					IF AR3SiSortedMasterTimeBlockFreeArmBuffer[iArmFL, iFreeSlotFL, 2] > 0 THEN
					AR3SiSortedMasterTimeBlockFreeArm_Out[iArmFL, ARiFreeSlotDataQtyArm_Out[iArmFL], 1] := AR3SiSortedMasterTimeBlockFreeArmBuffer[iArmFL, iFreeSlotFL, 1];
					AR3SiSortedMasterTimeBlockFreeArm_Out[iArmFL, ARiFreeSlotDataQtyArm_Out[iArmFL], 2] := AR3SiSortedMasterTimeBlockFreeArmBuffer[iArmFL, iFreeSlotFL, 2];
					AR3SiSortedMasterTimeBlockFreeArm_Out[iArmFL, ARiFreeSlotDataQtyArm_Out[iArmFL], 3] := AR3SiSortedMasterTimeBlockFreeArmBuffer[iArmFL, iFreeSlotFL, 3];
					ARiFreeSlotDataQtyArm_Out[iArmFL] := ARiFreeSlotDataQtyArm_Out[iArmFL] +1;
					ELSE
					AR3SiSortedMasterTimeBlockFreeArm_Out[iArmFL, iFreeSlotFL, 1] := 0;
					AR3SiSortedMasterTimeBlockFreeArm_Out[iArmFL, iFreeSlotFL, 2] := 0;
					AR3SiSortedMasterTimeBlockFreeArm_Out[iArmFL, iFreeSlotFL, 3] := 0;
					END_IF

				END_IF
			END_FOR
		END_IF
	END_FOR


(*fbV2_MTBConsolidateSorted - Clear Free Slot*)

	iStnFL := 1;
	FOR iStnFL := 1 TO iStnQty DO
		IF iStnFL >= 1 AND iStnFL <= iStnQty THEN
		iFreeSlotFL := 1;
		ARiFreeSlotDataQtyStn_Out[iStnFL] := 1;
			FOR iFreeSlotFL := 1 TO ARiFreeSlotDataQtyStn_in[iStnFL] DO
				IF iFreeSlotFL >= 1 AND iFreeSlotFL <= ARiFreeSlotDataQtyStn_in[iStnFL] THEN

					IF AR3SiSortedMasterTimeBlockFreeStnBuffer[iStnFL, iFreeSlotFL, 2] > 0 THEN
					AR3SiSortedMasterTimeBlockFreeStn_Out[iStnFL, ARiFreeSlotDataQtyStn_Out[iStnFL], 1] := AR3SiSortedMasterTimeBlockFreeStnBuffer[iStnFL, iFreeSlotFL, 1];
					AR3SiSortedMasterTimeBlockFreeStn_Out[iStnFL, ARiFreeSlotDataQtyStn_Out[iStnFL], 2] := AR3SiSortedMasterTimeBlockFreeStnBuffer[iStnFL, iFreeSlotFL, 2];
					AR3SiSortedMasterTimeBlockFreeStn_Out[iStnFL, ARiFreeSlotDataQtyStn_Out[iStnFL], 3] := AR3SiSortedMasterTimeBlockFreeStnBuffer[iStnFL, iFreeSlotFL, 3];
					ARiFreeSlotDataQtyStn_Out[iStnFL] := ARiFreeSlotDataQtyStn_Out[iStnFL] +1;
					ELSE
					AR3SiSortedMasterTimeBlockFreeStn_Out[iStnFL, iFreeSlotFL, 1] := 0;
					AR3SiSortedMasterTimeBlockFreeStn_Out[iStnFL, iFreeSlotFL, 2] := 0;
					AR3SiSortedMasterTimeBlockFreeStn_Out[iStnFL, iFreeSlotFL, 3] := 0;
					END_IF

				END_IF
			END_FOR
		END_IF
	END_FOR


(*fbV2_MTBConsolidateSorted - Clear Free Slot*)

	iUldFL := 1;
	FOR iUldFL := 1 TO iUldStnQty DO
		IF iUldFL >= 1 AND iUldFL <= iUldStnQty THEN
		iFreeSlotFL := 1;
		ARiFreeSlotDataQtyUld_Out[iUldFL] := 1;
			FOR iFreeSlotFL := 1 TO ARiFreeSlotDataQtyUld_in[iUldFL] DO
				IF iFreeSlotFL >= 1 AND iFreeSlotFL <= ARiFreeSlotDataQtyUld_in[iUldFL] THEN

					IF AR3SiSortedMasterTimeBlockFreeUldBuffer[iUldFL, iFreeSlotFL, 2] > 0 THEN
					AR3SiSortedMasterTimeBlockFreeUld_Out[iUldFL, ARiFreeSlotDataQtyUld_Out[iUldFL], 1] := AR3SiSortedMasterTimeBlockFreeUldBuffer[iUldFL, iFreeSlotFL, 1];
					AR3SiSortedMasterTimeBlockFreeUld_Out[iUldFL, ARiFreeSlotDataQtyUld_Out[iUldFL], 2] := AR3SiSortedMasterTimeBlockFreeUldBuffer[iUldFL, iFreeSlotFL, 2];
					AR3SiSortedMasterTimeBlockFreeUld_Out[iUldFL, ARiFreeSlotDataQtyUld_Out[iUldFL], 3] := AR3SiSortedMasterTimeBlockFreeUldBuffer[iUldFL, iFreeSlotFL, 3];
					ARiFreeSlotDataQtyUld_Out[iUldFL] := ARiFreeSlotDataQtyUld_Out[iUldFL] +1;
					ELSE
					AR3SiSortedMasterTimeBlockFreeUld_Out[iUldFL, iFreeSlotFL, 1] := 0;
					AR3SiSortedMasterTimeBlockFreeUld_Out[iUldFL, iFreeSlotFL, 2] := 0;
					AR3SiSortedMasterTimeBlockFreeUld_Out[iUldFL, iFreeSlotFL, 3] := 0;
					END_IF

				END_IF
			END_FOR
		END_IF
	END_FOR



(*
iStep := 13;
4:
*)
	iArmFL := 1;
	FOR iArmFL := 1 TO iArmQty DO
		IF iArmFL >= 1 AND iArmFL <= iArmQty THEN
			ARiFreeSlotDataQtyArm_Out[iArmFL] := ARiFreeSlotDataQtyArm_Out[iArmFL] -1;
		END_IF
	END_FOR

	iStnFL := 1;
	FOR iStnFL := 1 TO iStnQty DO
		IF iStnFL >= 1 AND iStnFL <= iStnQty THEN
			ARiFreeSlotDataQtyStn_Out[iStnFL] := ARiFreeSlotDataQtyStn_Out[iStnFL] -1;
		END_IF
	END_FOR


	iUldFL := 1;
	FOR iUldFL := 1 TO iUldStnQty DO
		IF iUldFL >= 1 AND iUldFL <= iUldStnQty THEN
			ARiFreeSlotDataQtyUld_Out[iUldFL] := ARiFreeSlotDataQtyUld_Out[iUldFL] -1;
		END_IF
	END_FOR

(*
iStep := 14;

11:;
12:;
13:;
14:;
15:;

END_CASE
*)
bDone := TRUE;
bEn := FALSE;
iPreviousShiftValue := iShiftValue;
END_IF

END_FUNCTION_BLOCK

// ---- FBs/B_JKS_NewFB_V2/FBP-MTBSubFB/fbV2_SubMTBFreeSlotGenerator.TcPOU
FUNCTION_BLOCK fbV2_SubMTBFreeSlotGenerator


(*************************************************************** Ver.B1 - fbV2_SubMTBFreeSlotGenerator - 160704 **************************************************************]

 	- Modify Search value to 20000 from 10000. Because the Add Value when the end block will be greater than 10000.																	
	- 
	- 	
	- 
[****************************************************************************************************************************************************************************************************)



VAR_INPUT
	bReset													: BOOL;
	AR3SiMTBBusyArm_In(*AR3SiMTBArm_In*) 					: ARRAY[1..iArmQty, 1..iMasterBlockQty, 1..3] OF INT;
	AR3SiMTBBusyStn_In(*AR3SiMTBStn_In*) 					: ARRAY[1..iStnQty, 1..iMasterBlockQty, 1..3] OF INT;
	AR3SiMTBBusyUld_In(*AR3SiMTBUld_In*) 					: ARRAY[1..iUldStnQty, 1..iMasterBlockQty, 1..3] OF INT;
	ARiArmID												: ARRAY [1..iArmQty] OF INT;
	ARiUldStnID												: ARRAY [1..iUldStnQty] OF INT;		(* To Define Unloading Station ID*)


END_VAR


VAR_IN_OUT
	bEn										: BOOL;

	AR3SiSortedMTBFreeArm_Out 				: ARRAY[1..iArmQty, 1..iMasterBlockQty, 1..3] OF INT;
	AR3SiSortedMTBFreeStn_Out 				: ARRAY[1..iStnQty, 1..iMasterBlockQty, 1..3] OF INT;
	AR3SiSortedMTBFreeUld_Out 				: ARRAY[1..iUldStnQty, 1..iMasterBlockQty, 1..3] OF INT;
	ARiMTBFreeSlotDataQtyArm				: ARRAY[1..iArmQty] OF INT;
	ARiMTBFreeSlotDataQtyStn				: ARRAY[1..iStnQty] OF INT;
	ARiMTBFreeSlotDataQtyUld				: ARRAY[1..iUldStnQty] OF INT;
END_VAR

VAR_OUTPUT
	bMTBEmpty : BOOL;
	bDone : BOOL;

END_VAR
VAR
	(*AR3SiMTBArm_Out*)AR3SiSortedMTBBusyArm(*_In*) 				: ARRAY[1..iArmQty, 1..iMasterBlockQty, 1..3] OF INT;
	(*AR3SiMTBStn_Out*)AR3SiSortedMTBBusyStn(*_In*) 				: ARRAY[1..iStnQty, 1..iMasterBlockQty, 1..3] OF INT;
	(*AR3SiMTBUld_Out*)AR3SiSortedMTBBusyUld(*_In*) 				: ARRAY[1..iUldStnQty, 1..iMasterBlockQty, 1..3] OF INT;

	(*ARiDataQtyArm*)ARiSortedDataQtyArm									: ARRAY[1..iArmQty] OF INT;
	(*ARiDataQtyStn*)ARiSortedDataQtyStn									: ARRAY[1..iStnQty] OF INT;
	(*ARiDataQtyUld*)ARiSortedDataQtyUld									: ARRAY[1..iUldStnQty] OF INT;

(****** From fbV2_MTBConsolidateSorted*)
	bResetRE: R_TRIG;

	bEnRE: R_TRIG;
	bEnFE: F_TRIG;
	iStep: INT;


	AR3SiBufferTimeBlockArm 						: ARRAY[1..iArmQty, 1..iMasterBlockQty, 1..3] OF INT;
	AR3SiBufferTimeBlockStn 						: ARRAY[1..iStnQty, 1..iMasterBlockQty, 1..3] OF INT;
	AR3SiBufferTimeBlockUld 						: ARRAY[1..iUldStnQty, 1..iMasterBlockQty, 1..3] OF INT;

	AR3SiBufferOrderArm	 						: ARRAY[1..iArmQty, 1..iMasterBlockQty] OF INT;
	AR3SiBufferOrderStn 							: ARRAY[1..iStnQty, 1..iMasterBlockQty] OF INT;
	AR3SiBufferOrderUld 							: ARRAY[1..iUldStnQty, 1..iMasterBlockQty] OF INT;

	AR3SiMTBArmEmpty 				: ARRAY[1..iArmQty, 1..iMasterBlockQty, 1..3] OF INT;
	AR3SiMTBStnEmpty 				: ARRAY[1..iStnQty, 1..iMasterBlockQty, 1..3] OF INT;
	AR3SiMTBUldEmpty 				: ARRAY[1..iUldStnQty, 1..iMasterBlockQty, 1..3] OF INT;

	AR3SiBufferOrderArmEmpty	 				: ARRAY[1..iArmQty, 1..iMasterBlockQty] OF INT;
	AR3SiBufferOrderStnEmpty	 					: ARRAY[1..iStnQty, 1..iMasterBlockQty] OF INT;
	AR3SiBufferOrderUldEmpty	 					: ARRAY[1..iUldStnQty, 1..iMasterBlockQty] OF INT;


	ARiCounterArmEmpty: ARRAY[1..iArmQty] OF INT;
	ARiCounterStnEmpty: ARRAY[1..iStnQty] OF INT;
	ARiCounterUldEmpty: ARRAY[1..iUldStnQty] OF INT;

	iSearchFL: INT;
	iSearchBuffer: INT;
	iSearchBufferAdd: INT;
	iSearchBufferValue: INT;
	iCounter: INT;
	iRunningNo: INT;

	iCheckFL: INT;
	iFreeSlotFL: INT;

	iArmFL: INT;
	iStnFL: INT;
	iUldFL: INT;

	ARiFoundCounterArm: ARRAY[1..iArmQty] OF INT;
	ARiFoundCounterStn: ARRAY[1..iStnQty] OF INT;
	ARiFoundCounterUld: ARRAY[1..iUldStnQty] OF INT;

	ARiScanCounterArm: ARRAY[1..iArmQty] OF INT;
	ARiScanCounterStn: ARRAY[1..iStnQty] OF INT;
	ARiScanCounterUld: ARRAY[1..iUldStnQty] OF INT;


	iGenFL: INT;
	iSkipArm: INT;
	iSkipStn: INT;
	iSkipUld: INT;
END_VAR

bResetRE(CLK:=bReset , Q=> );
bEnRE(CLK:=bEn , Q=> );

IF bResetRE.Q THEN
bDone := FALSE;
bMTBEmpty := FALSE;
END_IF

(*
IF NOT bEn THEN
bDone := FALSE;
END_IF
*)


IF NOT bReset AND bEnRE.Q THEN

	bDone := FALSE;
	bMTBEmpty := FALSE;
	iStep := 1;
	AR3SiSortedMTBBusyArm 				:= AR3SiMTBArmEmpty;
	AR3SiSortedMTBBusyStn 				:= AR3SiMTBStnEmpty;
	AR3SiSortedMTBBusyUld 				:= AR3SiMTBUldEmpty;

	AR3SiBufferOrderArm 					:= AR3SiBufferOrderArmEmpty;
	AR3SiBufferOrderStn 					:= AR3SiBufferOrderStnEmpty;
	AR3SiBufferOrderUld 					:= AR3SiBufferOrderUldEmpty;

	AR3SiBufferTimeBlockArm 				:= AR3SiMTBArmEmpty;
	AR3SiBufferTimeBlockStn 				:= AR3SiMTBStnEmpty;
	AR3SiBufferTimeBlockUld 				:= AR3SiMTBUldEmpty;

	ARiSortedDataQtyArm 					:= ARiCounterArmEmpty;
	ARiSortedDataQtyStn 					:= ARiCounterStnEmpty;
	ARiSortedDataQtyUld					:= ARiCounterUldEmpty;

	AR3SiSortedMTBFreeArm_Out 			:= AR3SiMTBArmEmpty;
	AR3SiSortedMTBFreeStn_Out 			:= AR3SiMTBStnEmpty;
	AR3SiSortedMTBFreeUld_Out 			:= AR3SiMTBUldEmpty;



END_IF

CASE iStep OF
0:;

1: (*fbV2_MTBConsolidateSorted - Clear Free Slot*)
	iArmFL := 1;
	FOR iArmFL := 1 TO iArmQty DO
		IF iArmFL >= 1 AND iArmFL <= iArmQty THEN
		iFreeSlotFL := 1;
		ARiSortedDataQtyArm[iArmFL] := 1;
			FOR iFreeSlotFL := 1 TO iMasterBlockQty DO
				IF iFreeSlotFL >= 1 AND iFreeSlotFL <= iMasterBlockQty THEN

					IF AR3SiMTBBusyArm_In[iArmFL, iFreeSlotFL, 2] > 0 THEN
					AR3SiBufferTimeBlockArm[iArmFL, ARiSortedDataQtyArm[iArmFL], 1] := AR3SiMTBBusyArm_In[iArmFL, iFreeSlotFL, 1];
					AR3SiBufferTimeBlockArm[iArmFL, ARiSortedDataQtyArm[iArmFL], 2] := AR3SiMTBBusyArm_In[iArmFL, iFreeSlotFL, 2];
					AR3SiBufferTimeBlockArm[iArmFL, ARiSortedDataQtyArm[iArmFL], 3] := AR3SiMTBBusyArm_In[iArmFL, iFreeSlotFL, 3];
					ARiSortedDataQtyArm[iArmFL] := ARiSortedDataQtyArm[iArmFL] +1;
					END_IF
				END_IF
			END_FOR
		END_IF
	END_FOR


	iStnFL := 1;
	FOR iStnFL := 1 TO iStnQty DO
		IF iStnFL >= 1 AND iStnFL <= iStnQty THEN
		iFreeSlotFL := 1;
		ARiSortedDataQtyStn[iStnFL] := 1;
			FOR iFreeSlotFL := 1 TO iMasterBlockQty DO
				IF iFreeSlotFL >= 1 AND iFreeSlotFL <= iMasterBlockQty THEN

					IF AR3SiMTBBusyStn_In[iStnFL, iFreeSlotFL, 2] > 0 THEN
					AR3SiBufferTimeBlockStn[iStnFL, ARiSortedDataQtyStn[iStnFL], 1] := AR3SiMTBBusyStn_In[iStnFL, iFreeSlotFL, 1];
					AR3SiBufferTimeBlockStn[iStnFL, ARiSortedDataQtyStn[iStnFL], 2] := AR3SiMTBBusyStn_In[iStnFL, iFreeSlotFL, 2];
					AR3SiBufferTimeBlockStn[iStnFL, ARiSortedDataQtyStn[iStnFL], 3] := AR3SiMTBBusyStn_In[iStnFL, iFreeSlotFL, 3];
					ARiSortedDataQtyStn[iStnFL] := ARiSortedDataQtyStn[iStnFL] +1;
					END_IF
				END_IF
			END_FOR
		END_IF
	END_FOR



	iUldFL := 1;
	FOR iUldFL := 1 TO iUldStnQty DO
		IF iUldFL >= 1 AND iUldFL <= iUldStnQty THEN
		iFreeSlotFL := 1;
		ARiSortedDataQtyUld[iUldFL] := 1;
			FOR iFreeSlotFL := 1 TO iMasterBlockQty DO
				IF iFreeSlotFL >= 1 AND iFreeSlotFL <= iMasterBlockQty THEN

					IF AR3SiMTBBusyUld_In[iUldFL, iFreeSlotFL, 2] > 0 THEN
					AR3SiBufferTimeBlockUld[iUldFL, ARiSortedDataQtyUld[iUldFL], 1] := AR3SiMTBBusyUld_In[iUldFL, iFreeSlotFL, 1];
					AR3SiBufferTimeBlockUld[iUldFL, ARiSortedDataQtyUld[iUldFL], 2] := AR3SiMTBBusyUld_In[iUldFL, iFreeSlotFL, 2];
					AR3SiBufferTimeBlockUld[iUldFL, ARiSortedDataQtyUld[iUldFL], 3] := AR3SiMTBBusyUld_In[iUldFL, iFreeSlotFL, 3];
					ARiSortedDataQtyUld[iUldFL] := ARiSortedDataQtyUld[iUldFL] +1;
					END_IF
				END_IF
			END_FOR
		END_IF
	END_FOR



	iArmFL := 1;
	FOR iArmFL := 1 TO iArmQty DO
		IF iArmFL >= 1 AND iArmFL <= iArmQty THEN
			ARiSortedDataQtyArm[iArmFL] := ARiSortedDataQtyArm[iArmFL] -1;
			ARiMTBFreeSlotDataQtyArm[iArmFL] := 0;
		END_IF
	END_FOR

	iStnFL := 1;
	FOR iStnFL := 1 TO iStnQty DO
		IF iStnFL >= 1 AND iStnFL <= iStnQty THEN
			ARiSortedDataQtyStn[iStnFL] := ARiSortedDataQtyStn[iStnFL] -1;
			ARiMTBFreeSlotDataQtyStn[iStnFL] := 0;
		END_IF
	END_FOR

	iUldFL := 1;
	FOR iUldFL := 1 TO iUldStnQty DO
		IF iUldFL >= 1 AND iUldFL <= iUldStnQty THEN
			ARiSortedDataQtyUld[iUldFL] := ARiSortedDataQtyUld[iUldFL] -1;
			ARiMTBFreeSlotDataQtyUld[iUldFL] := 0;
		END_IF
	END_FOR




iArmFL := 1;
iStnFL := 1;
iUldFL := 1;



iStep := 12;



12: (*fbV2_MTBConsolidateSorted - Data Sorting*)

	IF iArmFL <= iArmQty THEN
		ARiScanCounterArm[iArmFL] := 1;
		ARiFoundCounterArm[iArmFL] := 1;

		FOR ARiScanCounterArm[iArmFL] := 1 TO ARiSortedDataQtyArm[iArmFL] DO
			IF ARiScanCounterArm[iArmFL] >= 1 AND ARiScanCounterArm[iArmFL] <= ARiSortedDataQtyArm[iArmFL] THEN

				iSearchFL := 1;
				iSearchBufferValue := 20000;
				iSearchBufferAdd := 0;
					FOR iSearchFL := 1 TO ARiSortedDataQtyArm[iArmFL] DO
						IF iSearchFL >= 1 AND iSearchFL <= ARiSortedDataQtyArm[iArmFL] THEN

							IF AR3SiBufferOrderArm[iArmFL, iSearchFL] = 0 AND AR3SiBufferTimeBlockArm[iArmFL, iSearchFL, 2] > 0 THEN
								IF AR3SiBufferTimeBlockArm[iArmFL, iSearchFL, 2] <= iSearchBufferValue THEN
									iSearchBufferValue		:= AR3SiBufferTimeBlockArm[iArmFL, iSearchFL, 2];
									iSearchBufferAdd			:= iSearchFL;
								END_IF
							END_IF
						END_IF

					END_FOR

					IF iSearchFL > ARiSortedDataQtyArm[iArmFL] AND iSearchBufferAdd > 0 THEN
					AR3SiSortedMTBBusyArm[iArmFL, ARiFoundCounterArm[iArmFL], 1] := AR3SiBufferTimeBlockArm[iArmFL, iSearchBufferAdd, 1];
					AR3SiSortedMTBBusyArm[iArmFL, ARiFoundCounterArm[iArmFL], 2] := AR3SiBufferTimeBlockArm[iArmFL, iSearchBufferAdd, 2];
					AR3SiSortedMTBBusyArm[iArmFL, ARiFoundCounterArm[iArmFL], 3] := AR3SiBufferTimeBlockArm[iArmFL, iSearchBufferAdd, 3];
					AR3SiBufferOrderArm[iArmFL, iSearchBufferAdd] := ARiFoundCounterArm[iArmFL];
					ARiFoundCounterArm[iArmFL] := ARiFoundCounterArm[iArmFL] +1;
					END_IF

			END_IF
		END_FOR
	END_IF



	IF iStnFL <= iStnQty THEN
		ARiScanCounterStn[iStnFL] := 1;
		ARiFoundCounterStn[iStnFL] := 1;

		FOR ARiScanCounterStn[iStnFL] := 1 TO ARiSortedDataQtyStn[iStnFL] DO
			IF ARiScanCounterStn[iStnFL] >= 1 AND ARiScanCounterStn[iStnFL] <= ARiSortedDataQtyStn[iStnFL] THEN

				iSearchFL := 1;
				iSearchBufferValue := 20000;
				iSearchBufferAdd := 0;
					FOR iSearchFL := 1 TO ARiSortedDataQtyStn[iStnFL] DO
						IF iSearchFL >= 1 AND iSearchFL <= ARiSortedDataQtyStn[iStnFL] THEN

							IF AR3SiBufferOrderStn[iStnFL, iSearchFL] = 0 AND AR3SiBufferTimeBlockStn[iStnFL, iSearchFL, 2] > 0 THEN
								IF AR3SiBufferTimeBlockStn[iStnFL, iSearchFL, 2] <= iSearchBufferValue THEN
									iSearchBufferValue		:= AR3SiBufferTimeBlockStn[iStnFL, iSearchFL, 2];
									iSearchBufferAdd			:= iSearchFL;
								END_IF
							END_IF
						END_IF

					END_FOR

					IF iSearchFL > ARiSortedDataQtyStn[iStnFL] AND iSearchBufferAdd > 0 THEN
					AR3SiSortedMTBBusyStn[iStnFL, ARiFoundCounterStn[iStnFL], 1] := AR3SiBufferTimeBlockStn[iStnFL, iSearchBufferAdd, 1];
					AR3SiSortedMTBBusyStn[iStnFL, ARiFoundCounterStn[iStnFL], 2] := AR3SiBufferTimeBlockStn[iStnFL, iSearchBufferAdd, 2];
					AR3SiSortedMTBBusyStn[iStnFL, ARiFoundCounterStn[iStnFL], 3] := AR3SiBufferTimeBlockStn[iStnFL, iSearchBufferAdd, 3];
					AR3SiBufferOrderStn[iStnFL, iSearchBufferAdd] := ARiFoundCounterStn[iStnFL];
					ARiFoundCounterStn[iStnFL] := ARiFoundCounterStn[iStnFL] +1;
					END_IF

			END_IF
		END_FOR
	END_IF



	IF iUldFL <= iUldStnQty THEN
		ARiScanCounterUld[iUldFL] := 1;
		ARiFoundCounterUld[iUldFL] := 1;

		FOR ARiScanCounterUld[iUldFL] := 1 TO ARiSortedDataQtyUld[iUldFL] DO
			IF ARiScanCounterUld[iUldFL] >= 1 AND ARiScanCounterUld[iUldFL] <= ARiSortedDataQtyUld[iUldFL] THEN

				iSearchFL := 1;
				iSearchBufferValue := 20000;
				iSearchBufferAdd := 0;
					FOR iSearchFL := 1 TO ARiSortedDataQtyUld[iUldFL] DO
						IF iSearchFL >= 1 AND iSearchFL <= ARiSortedDataQtyUld[iUldFL] THEN

							IF AR3SiBufferOrderUld[iUldFL, iSearchFL] = 0 AND AR3SiBufferTimeBlockUld[iUldFL, iSearchFL, 2] > 0 THEN
								IF AR3SiBufferTimeBlockUld[iUldFL, iSearchFL, 2] <= iSearchBufferValue THEN
									iSearchBufferValue		:= AR3SiBufferTimeBlockUld[iUldFL, iSearchFL, 2];
									iSearchBufferAdd			:= iSearchFL;
								END_IF
							END_IF
						END_IF

					END_FOR

					IF iSearchFL > ARiSortedDataQtyUld[iUldFL] AND iSearchBufferAdd > 0 THEN
					AR3SiSortedMTBBusyUld[iUldFL, ARiFoundCounterUld[iUldFL], 1] := AR3SiBufferTimeBlockUld[iUldFL, iSearchBufferAdd, 1];
					AR3SiSortedMTBBusyUld[iUldFL, ARiFoundCounterUld[iUldFL], 2] := AR3SiBufferTimeBlockUld[iUldFL, iSearchBufferAdd, 2];
					AR3SiSortedMTBBusyUld[iUldFL, ARiFoundCounterUld[iUldFL], 3] := AR3SiBufferTimeBlockUld[iUldFL, iSearchBufferAdd, 3];
					AR3SiBufferOrderUld[iUldFL, iSearchBufferAdd] := ARiFoundCounterUld[iUldFL];
					ARiFoundCounterUld[iUldFL] := ARiFoundCounterUld[iUldFL] +1;
					END_IF

			END_IF
		END_FOR
	END_IF

iArmFL := iArmFL +1;
iStnFL := iStnFL +1;
iUldFL := iUldFL +1;

IF iArmFL > iArmQty AND iStnFL > iStnQty AND iUldFL > iUldStnQty THEN
iStep := 13;
END_IF

13:(*Generate FreeSlotBlock from Busy Block*)

	iArmFL := 1;
	iStnFL := 1;
	iUldFL := 1;

	FOR iArmFL := 1 TO iArmQty DO
		IF iArmFL >= 1 AND iArmFL <= iArmQty THEN
			iGenFL := 1;
			iSkipArm := 0;
			FOR iGenFL := 1 TO ARiSortedDataQtyArm[iArmFL] DO
				IF iGenFL >= 1 AND iGenFL <= ARiSortedDataQtyArm[iArmFL] THEN

					IF iGenFL = 1 THEN
						IF AR3SiSortedMTBBusyArm[iArmFL, iGenFL, 1] >1(*0*) THEN
							AR3SiSortedMTBFreeArm_Out[iArmFL, iGenFL, 1] := 0;
							AR3SiSortedMTBFreeArm_Out[iArmFL, iGenFL, 2] := AR3SiSortedMTBBusyArm[iArmFL, iGenFL, 1]-1;
							AR3SiSortedMTBFreeArm_Out[iArmFL, iGenFL, 3] := AR3SiSortedMTBBusyArm[iArmFL, iGenFL, 3];
							ARiMTBFreeSlotDataQtyArm[iArmFL] := ARiMTBFreeSlotDataQtyArm[iArmFL] +1;
						ELSE
							iSkipArm := 1;
						END_IF
					END_IF

					IF iGenFL >1 THEN
						IF AR3SiSortedMTBBusyArm[iArmFL, iGenFL, 1] >1(*0*) THEN
							AR3SiSortedMTBFreeArm_Out[iArmFL, iGenFL-iSkipArm, 1] := AR3SiSortedMTBBusyArm[iArmFL, iGenFL-1, 2]+1;
							AR3SiSortedMTBFreeArm_Out[iArmFL, iGenFL-iSkipArm, 2] := AR3SiSortedMTBBusyArm[iArmFL, iGenFL, 1]-1;
							AR3SiSortedMTBFreeArm_Out[iArmFL, iGenFL-iSkipArm, 3] := AR3SiSortedMTBBusyArm[iArmFL, iGenFL, 3];
							ARiMTBFreeSlotDataQtyArm[iArmFL] := ARiMTBFreeSlotDataQtyArm[iArmFL] +1;
						END_IF
					END_IF

					IF iGenFL =ARiSortedDataQtyArm[iArmFL] THEN
						IF AR3SiSortedMTBBusyArm[iArmFL, iGenFL, 2] >1(*0*) THEN
							AR3SiSortedMTBFreeArm_Out[iArmFL, iGenFL-iSkipArm+1, 1] := AR3SiSortedMTBBusyArm[iArmFL, iGenFL, 2]+1;
							AR3SiSortedMTBFreeArm_Out[iArmFL, iGenFL-iSkipArm+1, 2] := AR3SiSortedMTBBusyArm[iArmFL, iGenFL, 2]+1+10000;
							AR3SiSortedMTBFreeArm_Out[iArmFL, iGenFL-iSkipArm+1, 3] := AR3SiSortedMTBBusyArm[iArmFL, iGenFL, 3];
							ARiMTBFreeSlotDataQtyArm[iArmFL] := ARiMTBFreeSlotDataQtyArm[iArmFL] +1;
						END_IF
					END_IF
				END_IF
			END_FOR
		END_IF
	END_FOR


	FOR iStnFL := 1 TO iStnQty DO
		IF iStnFL >= 1 AND iStnFL <= iStnQty THEN
			iGenFL := 1;
			iSkipStn := 0;
			FOR iGenFL := 1 TO ARiSortedDataQtyStn[iStnFL] DO
				IF iGenFL >= 1 AND iGenFL <= ARiSortedDataQtyStn[iStnFL] THEN

					IF iGenFL = 1 THEN
						IF AR3SiSortedMTBBusyStn[iStnFL, iGenFL, 1] >1(*0*) THEN
							AR3SiSortedMTBFreeStn_Out[iStnFL, iGenFL, 1] := 0;
							AR3SiSortedMTBFreeStn_Out[iStnFL, iGenFL, 2] := AR3SiSortedMTBBusyStn[iStnFL, iGenFL, 1]-1;
							AR3SiSortedMTBFreeStn_Out[iStnFL, iGenFL, 3] := AR3SiSortedMTBBusyStn[iStnFL, iGenFL, 3];
							ARiMTBFreeSlotDataQtyStn[iStnFL] := ARiMTBFreeSlotDataQtyStn[iStnFL] +1;
						ELSE
							iSkipStn := 1;
						END_IF
					END_IF

					IF iGenFL >1 THEN
						IF AR3SiSortedMTBBusyStn[iStnFL, iGenFL, 1] >1(*0*) THEN
							AR3SiSortedMTBFreeStn_Out[iStnFL, iGenFL-iSkipStn, 1] := AR3SiSortedMTBBusyStn[iStnFL, iGenFL-1, 2]+1;
							AR3SiSortedMTBFreeStn_Out[iStnFL, iGenFL-iSkipStn, 2] := AR3SiSortedMTBBusyStn[iStnFL, iGenFL, 1]-1;
							AR3SiSortedMTBFreeStn_Out[iStnFL, iGenFL-iSkipStn, 3] := AR3SiSortedMTBBusyStn[iStnFL, iGenFL, 3];
							ARiMTBFreeSlotDataQtyStn[iStnFL] := ARiMTBFreeSlotDataQtyStn[iStnFL] +1;
						END_IF
					END_IF

					IF iGenFL =ARiSortedDataQtyStn[iStnFL] THEN
						IF AR3SiSortedMTBBusyStn[iStnFL, iGenFL, 2] >1(*0*) THEN
							AR3SiSortedMTBFreeStn_Out[iStnFL, iGenFL-iSkipStn+1, 1] := AR3SiSortedMTBBusyStn[iStnFL, iGenFL, 2]+1;
							AR3SiSortedMTBFreeStn_Out[iStnFL, iGenFL-iSkipStn+1, 2] := AR3SiSortedMTBBusyStn[iStnFL, iGenFL, 2]+1+10000;
							AR3SiSortedMTBFreeStn_Out[iStnFL, iGenFL-iSkipStn+1, 3] := AR3SiSortedMTBBusyStn[iStnFL, iGenFL, 3];
							ARiMTBFreeSlotDataQtyStn[iStnFL] := ARiMTBFreeSlotDataQtyStn[iStnFL] +1;
						END_IF
					END_IF
				END_IF
			END_FOR
		END_IF
	END_FOR



	FOR iUldFL := 1 TO iUldStnQty DO
		IF iUldFL >= 1 AND iUldFL <= iUldStnQty THEN
			iGenFL := 1;
			iSkipUld := 0;
			FOR iGenFL := 1 TO ARiSortedDataQtyUld[iUldFL] DO
				IF iGenFL >= 1 AND iGenFL <= ARiSortedDataQtyUld[iUldFL] THEN

					IF iGenFL = 1 THEN
						IF AR3SiSortedMTBBusyUld[iUldFL, iGenFL, 1] >1(*0*) THEN
							AR3SiSortedMTBFreeUld_Out[iUldFL, iGenFL, 1] := 0;
							AR3SiSortedMTBFreeUld_Out[iUldFL, iGenFL, 2] := AR3SiSortedMTBBusyUld[iUldFL, iGenFL, 1]-1;
							AR3SiSortedMTBFreeUld_Out[iUldFL, iGenFL, 3] := AR3SiSortedMTBBusyUld[iUldFL, iGenFL, 3];
							ARiMTBFreeSlotDataQtyUld[iUldFL] := ARiMTBFreeSlotDataQtyUld[iUldFL] +1;
						ELSE
							iSkipUld := 1;
						END_IF
					END_IF

					IF iGenFL >1 THEN
						IF AR3SiSortedMTBBusyUld[iUldFL, iGenFL, 1] >1(*0*) THEN
							AR3SiSortedMTBFreeUld_Out[iUldFL, iGenFL-iSkipUld, 1] := AR3SiSortedMTBBusyUld[iUldFL, iGenFL-1, 2]+1;
							AR3SiSortedMTBFreeUld_Out[iUldFL, iGenFL-iSkipUld, 2] := AR3SiSortedMTBBusyUld[iUldFL, iGenFL, 1]-1;
							AR3SiSortedMTBFreeUld_Out[iUldFL, iGenFL-iSkipUld, 3] := AR3SiSortedMTBBusyUld[iUldFL, iGenFL, 3];
							ARiMTBFreeSlotDataQtyUld[iUldFL] := ARiMTBFreeSlotDataQtyUld[iUldFL] +1;
						END_IF
					END_IF

					IF iGenFL =ARiSortedDataQtyUld[iUldFL] THEN
						IF AR3SiSortedMTBBusyUld[iUldFL, iGenFL, 2] >1(*0*) THEN
							AR3SiSortedMTBFreeUld_Out[iUldFL, iGenFL-iSkipUld+1, 1] := AR3SiSortedMTBBusyUld[iUldFL, iGenFL, 2]+1;
							AR3SiSortedMTBFreeUld_Out[iUldFL, iGenFL-iSkipUld+1, 2] := AR3SiSortedMTBBusyUld[iUldFL, iGenFL, 2]+1+10000;
							AR3SiSortedMTBFreeUld_Out[iUldFL, iGenFL-iSkipUld+1, 3] := AR3SiSortedMTBBusyUld[iUldFL, iGenFL, 3];
							ARiMTBFreeSlotDataQtyUld[iUldFL] := ARiMTBFreeSlotDataQtyUld[iUldFL] +1;
						END_IF
					END_IF
				END_IF
			END_FOR
		END_IF
	END_FOR




iStep:= 14;

14: (* Put Remark for those "0" = "Empty" Stn *) (*Generate FreeSlotBlock for Empty Stn Block*)

bMTBEmpty := TRUE;

	iArmFL := 1;
	FOR iArmFL := 1 TO iArmQty DO
		IF iArmFL >= 1 AND iArmFL <= iArmQty THEN

			IF ARiMTBFreeSlotDataQtyArm[iArmFL] > 0 THEN
				bMTBEmpty := FALSE;
			END_IF

			IF ARiMTBFreeSlotDataQtyArm[iArmFL] = 0 THEN
				AR3SiSortedMTBFreeArm_Out[iArmFL, 1, 1] := 0;
				AR3SiSortedMTBFreeArm_Out[iArmFL, 1, 2] := 10000;
				AR3SiSortedMTBFreeArm_Out[iArmFL, 1, 3] := ARiArmID[iArmFL];
				ARiMTBFreeSlotDataQtyArm[iArmFL] := 1;
			END_IF
		END_IF
	END_FOR


	iStnFL := 1;
	FOR iStnFL := 1 TO iStnQty DO
		IF iStnFL >= 1 AND iStnFL <= iStnQty THEN

			IF ARiMTBFreeSlotDataQtyStn[iStnFL] > 0 THEN
				bMTBEmpty := FALSE;
			END_IF

			IF ARiMTBFreeSlotDataQtyStn[iStnFL] = 0 THEN
				AR3SiSortedMTBFreeStn_Out[iStnFL, 1, 1] := 0;
				AR3SiSortedMTBFreeStn_Out[iStnFL, 1, 2] := 10000;
				AR3SiSortedMTBFreeStn_Out[iStnFL, 1, 3] := iStnFL;
				ARiMTBFreeSlotDataQtyStn[iStnFL] := 1;
			END_IF
		END_IF
	END_FOR


	iUldFL := 1;
	FOR iUldFL := 1 TO iUldStnQty DO
		IF iUldFL >= 1 AND iUldFL <= iUldStnQty THEN

			IF ARiMTBFreeSlotDataQtyUld[iUldFL] > 0 THEN
				bMTBEmpty := FALSE;
			END_IF

			IF ARiMTBFreeSlotDataQtyUld[iUldFL] = 0 THEN
				AR3SiSortedMTBFreeUld_Out[iUldFL, 1, 1] := 0;
				AR3SiSortedMTBFreeUld_Out[iUldFL, 1, 2] := 10000;
				AR3SiSortedMTBFreeUld_Out[iUldFL, 1, 3] := ARiUldStnID[iUldFL];
				ARiMTBFreeSlotDataQtyUld[iUldFL] := 1;
			END_IF
		END_IF
	END_FOR

iStep := 20;


20: (* Search Completed*)
bDone := TRUE;
bEn := FALSE;


END_CASE

END_FUNCTION_BLOCK

// ---- FBs/B_JKS_NewFB_V2/FBP-MTBSubFB/fbV2_SubMTBRTBCrashCheck.TcPOU
FUNCTION_BLOCK fbV2_SubMTBRTBCrashCheck
VAR_INPUT
	bEn										: BOOL;
	bReset									: BOOL;
	bBusyLinkMasterCheck					: BOOL;
	bBusyLinkSlaveCheck						: BOOL;
	iCurrentMasterFreeBlockStart 				: INT; 	(*MD1*)		(*Array "1"*)
	iCurrentMasterFreeBlockEnd 				: INT;	(*MD2*)		(*Array "2"*)
(*	iNextMasterFreeBlockStart 					: INT; 	(*MD3*)
	iNextMasterFreeBlockEnd 					: INT;	(*MD4*)
*)	iCurrentRecipeBusyBlockStart 				: INT;	(*RD1*)		(*Array "1"*)
	iCurrentRecipeBusyBlockEnd 				: INT;	(*RD2*)		(*Array "2"*)
	iCurrentRecipeBusyTime					: INT;				(*Array "5"*)
	iCurrentRecipeBusyBlockMinTime			: INT;				(*Array "6"*)
	iCurrentRecipeBusyBlockMaxTime			: INT;				(*Array "7"*)
	iCurrentRecipeBusyLinkMasterSlaveAdd		: INT;				(*Array "9"*)
	iCurrentShiftAllowedTime					: INT; 	(*Determine by Previous Station Remained Tolerance Time VS Crashed Time Whichever Lower*)

END_VAR
VAR_IN_OUT
	iMTB_NATime							: INT;
END_VAR

VAR_OUTPUT

(**)	bMTB_ShiftBlockRequestFlag	: BOOL; (*Current Master Time Block Empty or Not Suitable for Scanning Used, Out of range*)
(**)	bRTB_ShiftBlockRequestFlag	: BOOL; (*Current Recipe Time Block Empty*)
(**)	bSpacingOK 					: BOOL;
(**)	bNoCrashFound				: BOOL;
(**)	iNextShiftAllowedTime			: INT;	(*Determine Balance Time for Next Block Shifting Based on Remained Tolerance Time VS Crashed Time whichever lower*)

(**)	bSpacingNG 					: BOOL;
	bCrashFound 				: BOOL;

(**)	bMTB_ShiftTimeRequestFlag 	: BOOL;
(**)	iMTB_ShiftTime	 			: INT;

(**)	bRTB_ShiftTimeRequestFlag 	: BOOL;
(**)	iRTB_ShiftTime	 			: INT;

	bBusyLinkMasterSkipFlag		: BOOL;
	bBusyLinkSlaveSkipFlag		: BOOL;

	bError						: BOOL;


END_VAR
VAR

	bEnFE: F_TRIG;
	iCurrentRecipeBusyBlockTolerance	: INT;

	iExtTime: INT;
	bResetRE: R_TRIG;
END_VAR

bResetRE(CLK:=bReset , Q=> );

IF bResetRE.Q THEN
	bMTB_ShiftBlockRequestFlag	:= FALSE;
	bRTB_ShiftBlockRequestFlag	:= FALSE;

	bSpacingOK 					:= FALSE;
	bNoCrashFound				:= FALSE;
	iNextShiftAllowedTime 			:= 0;

	bSpacingNG 					:= FALSE;
	bCrashFound 				:= FALSE;

	bMTB_ShiftTimeRequestFlag 	:= FALSE;
	iMTB_ShiftTime	 			:= 0;

	bRTB_ShiftTimeRequestFlag 	:= FALSE;
	iRTB_ShiftTime	 			:= 0;

	bBusyLinkMasterSkipFlag		:= FALSE;
	bBusyLinkSlaveSkipFlag		:= FALSE;
	bError						:= FALSE;

END_IF


IF bEn THEN

(*Initialised*)
	bMTB_ShiftBlockRequestFlag	:= FALSE;
	bRTB_ShiftBlockRequestFlag	:= FALSE;

	bSpacingOK 					:= FALSE;
	bNoCrashFound				:= FALSE;
	iNextShiftAllowedTime 			:= 0;

	bSpacingNG 					:= FALSE;
	bCrashFound 				:= FALSE;

	bMTB_ShiftTimeRequestFlag 	:= FALSE;
	iMTB_ShiftTime	 			:= 0;

	bRTB_ShiftTimeRequestFlag 	:= FALSE;
	iRTB_ShiftTime	 			:= 0;

	bBusyLinkMasterSkipFlag		:= FALSE;
	bBusyLinkSlaveSkipFlag		:= FALSE;
	bError						:= FALSE;



(*Checking / Scanning Start*)

	(*Check BusyLink Master And Slave Operation*)
	IF bBusyLinkMasterCheck AND iCurrentRecipeBusyLinkMasterSlaveAdd > 99 THEN
		bBusyLinkSlaveSkipFlag := TRUE;
	ELSIF bBusyLinkSlaveCheck AND iCurrentRecipeBusyLinkMasterSlaveAdd <100 THEN
		bBusyLinkMasterSkipFlag := TRUE;

	(*RTB Empty / Error Block - Cannot Scan*)
	ELSIF (iCurrentRecipeBusyBlockEnd (*RD2*)  <= 0)									(*Empty Block*)
		OR (iCurrentRecipeBusyBlockStart (*RD1*) >= iCurrentRecipeBusyBlockEnd (*RD2*))	(*Error Block*)
		THEN

		bRTB_ShiftBlockRequestFlag	:= TRUE;
		bError						:= TRUE;


	(*MTB Empty / Error - Cannot Scan*)

	ELSIF (iCurrentMasterFreeBlockEnd (*MD2*)  <= 0)									(*Empty Block*)
		OR( (iCurrentMasterFreeBlockStart (*MD1*) ) - (iCurrentMasterFreeBlockEnd (*MD2*))) > 1		(*Error Block*)
		(*OR (iCurrentMasterFreeBlockEnd (*MD2*) <= iCurrentRecipeBusyBlockStart (*RD1*))		(*Not Suitable Block*)*)
		THEN

		bMTB_ShiftBlockRequestFlag	:= TRUE;
		bError						:= TRUE;


	(*MTB Not Suitable Block - Cannot Scan*)

	ELSIF (iCurrentMasterFreeBlockEnd (*MD2*) <= iCurrentRecipeBusyBlockStart (*RD1*))		(*Not Suitable Block*)
		THEN

		bMTB_ShiftBlockRequestFlag	:= TRUE;

	ELSE
	
		(*Check is Spacing OK or NG*)
		IF (iCurrentMasterFreeBlockEnd (*MD2*) - iCurrentMasterFreeBlockStart (*MD1*)+1) >= (iCurrentRecipeBusyBlockEnd (*RD2*) - iCurrentRecipeBusyBlockStart (*RD1*)+1) THEN
			bSpacingOK := TRUE;
		ELSE
			bSpacingNG := TRUE;
		END_IF
	
		(*Spacing OK & RTB Able to Fill into MTB without issue*)
		IF bSpacingOK
			AND (iCurrentMasterFreeBlockStart (*MD1*) <= iCurrentRecipeBusyBlockStart (*RD1*) AND iCurrentMasterFreeBlockEnd (*MD2*) >= iCurrentRecipeBusyBlockEnd (*RD2*))
			THEN
			bNoCrashFound 				:= TRUE;
			bRTB_ShiftBlockRequestFlag	:= TRUE;

				IF iMTB_NATime >  (iCurrentMasterFreeBlockEnd (*MD2*) - iCurrentRecipeBusyBlockEnd (*RD2*)) THEN
					iMTB_NATime := (iCurrentMasterFreeBlockEnd (*MD2*) - iCurrentRecipeBusyBlockEnd (*RD2*));
				END_IF

				IF (iCurrentRecipeBusyBlockMaxTime - iCurrentRecipeBusyBlockMinTime) <= 0 THEN
	
					IF iCurrentShiftAllowedTime >= (iCurrentMasterFreeBlockEnd (*MD2*) - iCurrentRecipeBusyBlockEnd (*RD2*)) THEN
					iNextShiftAllowedTime := (iCurrentMasterFreeBlockEnd (*MD2*) - iCurrentRecipeBusyBlockEnd (*RD2*));
					ELSE
					iNextShiftAllowedTime := iCurrentShiftAllowedTime;
					END_IF
		
				ELSE
		
					iExtTime := ((iCurrentRecipeBusyBlockEnd (*RD2*) - iCurrentRecipeBusyBlockStart (*RD1*)+1) - iCurrentRecipeBusyTime);
		
					IF ((iCurrentRecipeBusyBlockMaxTime - iCurrentRecipeBusyBlockMinTime) - iExtTime) >= (iCurrentMasterFreeBlockEnd (*MD2*) - iCurrentRecipeBusyBlockEnd (*RD2*)) THEN
					iNextShiftAllowedTime := (iCurrentMasterFreeBlockEnd (*MD2*) - iCurrentRecipeBusyBlockEnd (*RD2*));
					ELSE
		
						IF ((iCurrentRecipeBusyBlockMaxTime - iCurrentRecipeBusyBlockMinTime) - iExtTime) > 0 THEN
						iNextShiftAllowedTime := ((iCurrentRecipeBusyBlockMaxTime - iCurrentRecipeBusyBlockMinTime) - iExtTime);
						ELSE
						iNextShiftAllowedTime := 0;
						END_IF
		
		
					END_IF
	
				END_IF
		
		(*Spacing OK and check whether shifting is enough*)
		ELSIF bSpacingOK
			AND (iCurrentMasterFreeBlockStart (*MD1*) >= iCurrentRecipeBusyBlockStart (*RD1*) AND iCurrentMasterFreeBlockEnd (*MD2*) >= iCurrentRecipeBusyBlockEnd (*RD2*))
			THEN
				bCrashFound := TRUE;

					IF iCurrentShiftAllowedTime >= (iCurrentMasterFreeBlockStart (*MD1*) - iCurrentRecipeBusyBlockStart (*RD1*)) AND bBusyLinkMasterCheck THEN
					iRTB_ShiftTime := (iCurrentMasterFreeBlockStart (*MD1*) - iCurrentRecipeBusyBlockStart (*RD1*));
					bRTB_ShiftTimeRequestFlag := TRUE;
					ELSE
					iMTB_ShiftTime := (iCurrentMasterFreeBlockStart (*MD1*) - iCurrentRecipeBusyBlockStart (*RD1*));
					bMTB_ShiftTimeRequestFlag := TRUE;
					END_IF
		
	
		ELSE
			bMTB_ShiftBlockRequestFlag	:= TRUE;
		END_IF

	END_IF

END_IF

END_FUNCTION_BLOCK

// ---- FBs/B_JKS_NewFB_V2/FBP-MTBSubFB/fbV2_SubMTBRunningTime.TcPOU
FUNCTION_BLOCK fbV2_SubMTBRunningTime
VAR_INPUT
	bStart 																		: BOOL;
	bHalt 																		: BOOL;
	bReset 																		: BOOL;
	bCopyBusyToFreeMTB														: BOOL;
	bWrite_RTBtoMTB															: BOOL;
	iLoadingCallArmTime	 														: INT;
	AR2SiRecipeTimeBlockWithCallArmTime 										: ARRAY[1..iRecipeBlockQty, 1..9] OF INT;
	ARbAlternateStnEn 															: ARRAY [1..iAlternateSetQty] OF BOOL;
	AR2siAlternateStn 																: ARRAY [1..iAlternateSetQty, 1..iAlternateStnQty] OF INT;
	ARiArmID																	: ARRAY [1..iArmQty] OF INT;
	ARiUldStnID																	: ARRAY [1..iUldStnQty] OF INT;		(* To Define Unloading Station ID*)
(*
	iRTBScanBlockNo															: INT;
*)
END_VAR

VAR_OUTPUT
	bBusy 														 : BOOL;
	ARbArmProgress												 : ARRAY [1..iArmQty] OF BOOL;
	bCopyDone													: BOOL;
	bCopiedMTBEmptyFlag										: BOOL;

	bWriteBusy													 : BOOL;
	bWriteDone 													 : BOOL;
	bWriteMTBArmBlockFullError									 : BOOL;
	bWriteMTBStnBlockFullError									 : BOOL;
	bWriteMTBUldBlockFullError									 : BOOL;

	diSinceStartRunningTime										 : DINT;
	diSinceCopyRunningTime										 : DINT;

END_VAR

VAR
	tWriteDoneTimer									: TON;
	tOneSecClockPulse								: TON;

	tOneSecClockPulseRE								: R_TRIG;
	bResetRE										: R_TRIG;
	bCopyMTBRE									: R_TRIG;
	bWrite_RTBtoMTBRE								: R_TRIG;

	AR3SiMTBBusyArm_Empty				: ARRAY[1..iArmQty, 1..iMasterBlockQty, 1..3] OF INT;
	AR3SiMTBBusyStn_Empty		 		: ARRAY[1..iStnQty, 1..iMasterBlockQty, 1..3] OF INT;
	AR3SiMTBBusyUld_Empty 				: ARRAY[1..iUldStnQty, 1..iMasterBlockQty, 1..3] OF INT;

	AR2SiRecipeTimeBlockNoCallArmTime 				: ARRAY[1..iRecipeBlockQty, 1..9] OF INT;

	fbV2SubRTBGenerateNoCallArmTime				: fbV2_SubRTBGenerateNoCallArmTime;
	fbV2SubRTBEndStepFinder						: fbV2_SubRTBEndStepFinder;
	fbV2SubRTBStnTypeAltIDFinder					: fbV2_SubRTBStnTypeAltIDFinder;


	bEndStepFinderEn: BOOL;
	bEndStepFinderDone: BOOL;
	bEndStepFinderReset: BOOL;
	bNoCallArmTimeReset: BOOL;
	bNoCallArmTimeDone: BOOL;
	bNoCallArmTimeEn: BOOL;

	bFBEn 					: ARRAY [1..10] OF BOOL;
	bFBDone 				: ARRAY [1..10] OF BOOL;
	bFBReset 				: ARRAY [1..10] OF BOOL;
	bFBBusy 				: ARRAY [1..10] OF BOOL;

	iWriteStep: INT;
	iRTBEndStep: INT;

	iWriteMFL								: INT;
	iWriteSFL								: INT;

	bWriteArmDone							: BOOL;
	bWriteStnDone							: BOOL;
	bWriteUldDone							: BOOL;


(*fbV2SubRTBStnTypeAltIDFinder Used*)
	bRTBEmptyBlockFound					: BOOL;
	bRTBArmIDFound							: BOOL;
	bRTBStnIDFound							: BOOL;
	bRTBUldIDFound							: BOOL;
	bRTBAltStnIDFound						: BOOL;
	iRTBArmAdd								: INT;
	iRTBStnAdd								: INT;
	iRTBUldAdd								: INT;
	ARiRTBAltStnIDFound						: ARRAY [1..iAlternateStnQty] OF INT;
	ARiRTBAltStnAddFound					: ARRAY [1..iAlternateStnQty] OF INT;

	bMinusOneSecSt: BOOL;
	iMinusOneArmMFL: INT;
	iMinusOneStnMFL: INT;
	iMinusOneUldMFL: INT;
	iMinusOneArmSFL: INT;
	iMinusOneStnSFL: INT;
	iMinusOneUldSFL: INT;
	iArmProgressClearFL: INT;
	bMinusOneSecStRE: R_TRIG;
	fbV2SubMTBFreeSlotGenerator: fbV2_SubMTBFreeSlotGenerator;
	bConvertBusyToFreeMTBRE: R_TRIG;
	bCopyBusyToFreeMTBRE: R_TRIG;
	bWaitForReset: BOOL;
END_VAR

VAR_IN_OUT
	AR3SiMTBBusyArm_Main 										: ARRAY[1..iArmQty, 1..iMasterBlockQty, 1..3] OF INT;
	AR3SiMTBBusyStn_Main 										: ARRAY[1..iStnQty, 1..iMasterBlockQty, 1..3] OF INT;
	AR3SiMTBBusyUld_Main 										: ARRAY[1..iUldStnQty, 1..iMasterBlockQty, 1..3] OF INT;
	AR3SiSortedMTBFreeArm_Out									: ARRAY[1..iArmQty, 1..iMasterBlockQty, 1..3] OF INT;
	AR3SiSortedMTBFreeStn_Out									: ARRAY[1..iStnQty, 1..iMasterBlockQty, 1..3] OF INT;
	AR3SiSortedMTBFreeUld_Out									: ARRAY[1..iUldStnQty, 1..iMasterBlockQty, 1..3] OF INT;
	ARiMTBFreeSlotDataQtyArm									: ARRAY[1..iArmQty] OF INT;
	ARiMTBFreeSlotDataQtyStn									: ARRAY[1..iStnQty] OF INT;
	ARiMTBFreeSlotDataQtyUld									: ARRAY[1..iUldStnQty] OF INT;

END_VAR

tOneSecClockPulse			(IN:=NOT tOneSecClockPulse.Q , 	PT:=t#1s , Q=> , ET=> );
tWriteDoneTimer				(IN:=iWriteStep = 4 , 				PT:=t#0.5s , Q=> , ET=> );

tOneSecClockPulseRE			(CLK:=tOneSecClockPulse.Q , 				Q=> );
bResetRE					(CLK:=bReset , 							Q=> );
bCopyBusyToFreeMTBRE		(CLK:=bCopyBusyToFreeMTB , 				Q=> );
bWrite_RTBtoMTBRE			(CLK:=bWrite_RTBtoMTB , 					Q=> );
bMinusOneSecStRE			(CLK:=bMinusOneSecSt , 					Q=> );





(*Running Time*)
IF bStart AND NOT bHalt AND NOT bReset THEN
	bBusy := TRUE;
	IF tOneSecClockPulseRE.Q THEN
		diSinceCopyRunningTime := diSinceCopyRunningTime +1;
		diSinceStartRunningTime := diSinceStartRunningTime +1;
		bMinusOneSecSt := TRUE;
	END_IF
ELSE
	bBusy := FALSE;
	bMinusOneSecSt := FALSE;


	iArmProgressClearFL := 1;
	FOR iArmProgressClearFL := 1 TO iArmQty DO
		IF iArmProgressClearFL >= 1 AND iArmProgressClearFL <= iArmQty THEN
		ARbArmProgress[iArmProgressClearFL] := FALSE;
		END_IF
	END_FOR

END_IF

(*MTB - Minus One Sec*)
IF bMinusOneSecStRE.Q THEN


	(*Arm Section*)
	iMinusOneArmMFL := 1;
	FOR iMinusOneArmMFL := 1 TO iArmQty DO
		IF iMinusOneArmMFL >= 1 AND iMinusOneArmMFL <= iArmQty THEN

			ARbArmProgress[iMinusOneArmMFL] := FALSE;

			iMinusOneArmSFL := 1;
			FOR iMinusOneArmSFL := 1 TO iMasterBlockQty DO
				IF iMinusOneArmSFL >= 1 AND iMinusOneArmSFL <= iMasterBlockQty THEN

					IF AR3SiMTBBusyArm_Main[iMinusOneArmMFL, iMinusOneArmSFL, 1] > 0 THEN
					AR3SiMTBBusyArm_Main[iMinusOneArmMFL, iMinusOneArmSFL, 1] := AR3SiMTBBusyArm_Main[iMinusOneArmMFL, iMinusOneArmSFL, 1] -1;
					END_IF

					IF AR3SiMTBBusyArm_Main[iMinusOneArmMFL, iMinusOneArmSFL, 2] > 0 THEN
					AR3SiMTBBusyArm_Main[iMinusOneArmMFL, iMinusOneArmSFL, 2] := AR3SiMTBBusyArm_Main[iMinusOneArmMFL, iMinusOneArmSFL, 2] -1;
					ELSE
					AR3SiMTBBusyArm_Main[iMinusOneArmMFL, iMinusOneArmSFL, 1] := 0;
					AR3SiMTBBusyArm_Main[iMinusOneArmMFL, iMinusOneArmSFL, 2] := 0;
					AR3SiMTBBusyArm_Main[iMinusOneArmMFL, iMinusOneArmSFL, 3] := 0;
					END_IF

					IF AR3SiMTBBusyArm_Main[iMinusOneArmMFL, iMinusOneArmSFL, 1] = 0 AND AR3SiMTBBusyArm_Main[iMinusOneArmMFL, iMinusOneArmSFL, 2] > 0	 THEN
					ARbArmProgress[iMinusOneArmMFL] := TRUE;
					END_IF

				END_IF
			END_FOR
		END_IF
	END_FOR


	(*Stn Section*)
	iMinusOneStnMFL := 1;
	FOR iMinusOneStnMFL := 1 TO iStnQty DO
		IF iMinusOneStnMFL >= 1 AND iMinusOneStnMFL <= iStnQty THEN

			iMinusOneStnSFL := 1;
			FOR iMinusOneStnSFL := 1 TO iMasterBlockQty DO
				IF iMinusOneStnSFL >= 1 AND iMinusOneStnSFL <= iMasterBlockQty THEN

					IF AR3SiMTBBusyStn_Main[iMinusOneStnMFL, iMinusOneStnSFL, 1] > 0 THEN
					AR3SiMTBBusyStn_Main[iMinusOneStnMFL, iMinusOneStnSFL, 1] := AR3SiMTBBusyStn_Main[iMinusOneStnMFL, iMinusOneStnSFL, 1] -1;
					END_IF

					IF AR3SiMTBBusyStn_Main[iMinusOneStnMFL, iMinusOneStnSFL, 2] > 0 THEN
					AR3SiMTBBusyStn_Main[iMinusOneStnMFL, iMinusOneStnSFL, 2] := AR3SiMTBBusyStn_Main[iMinusOneStnMFL, iMinusOneStnSFL, 2] -1;
					ELSE
					AR3SiMTBBusyStn_Main[iMinusOneStnMFL, iMinusOneStnSFL, 1] := 0;
					AR3SiMTBBusyStn_Main[iMinusOneStnMFL, iMinusOneStnSFL, 2] := 0;
					AR3SiMTBBusyStn_Main[iMinusOneStnMFL, iMinusOneStnSFL, 3] := 0;
					END_IF

				END_IF
			END_FOR
		END_IF
	END_FOR


	(*Uld Section*)
	iMinusOneUldMFL := 1;
	FOR iMinusOneUldMFL := 1 TO iUldStnQty DO
		IF iMinusOneUldMFL >= 1 AND iMinusOneUldMFL <= iUldStnQty THEN

			iMinusOneUldSFL := 1;
			FOR iMinusOneUldSFL := 1 TO iMasterBlockQty DO
				IF iMinusOneUldSFL >= 1 AND iMinusOneUldSFL <= iMasterBlockQty THEN

					IF AR3SiMTBBusyUld_Main[iMinusOneUldMFL, iMinusOneUldSFL, 1] > 0 THEN
					AR3SiMTBBusyUld_Main[iMinusOneUldMFL, iMinusOneUldSFL, 1] := AR3SiMTBBusyUld_Main[iMinusOneUldMFL, iMinusOneUldSFL, 1] -1;
					END_IF

					IF AR3SiMTBBusyUld_Main[iMinusOneUldMFL, iMinusOneUldSFL, 2] > 0 THEN
					AR3SiMTBBusyUld_Main[iMinusOneUldMFL, iMinusOneUldSFL, 2] := AR3SiMTBBusyUld_Main[iMinusOneUldMFL, iMinusOneUldSFL, 2] -1;
					ELSE
					AR3SiMTBBusyUld_Main[iMinusOneUldMFL, iMinusOneUldSFL, 1] := 0;
					AR3SiMTBBusyUld_Main[iMinusOneUldMFL, iMinusOneUldSFL, 2] := 0;
					AR3SiMTBBusyUld_Main[iMinusOneUldMFL, iMinusOneUldSFL, 3] := 0;
					END_IF

				END_IF
			END_FOR
		END_IF
	END_FOR

bMinusOneSecSt := FALSE;

END_IF


(*MTB Reset*)
IF bResetRE.Q THEN
	AR3SiMTBBusyArm_Main 		:=	AR3SiMTBBusyArm_Empty;
	AR3SiMTBBusyStn_Main 		:=	AR3SiMTBBusyStn_Empty;
	AR3SiMTBBusyUld_Main 		:=	AR3SiMTBBusyUld_Empty;
	diSinceStartRunningTime := 0;
	diSinceCopyRunningTime := 0;
END_IF


(***************************************************************** MTB Copy *******************************************************************************)
(*MTB Copy*)
IF NOT bCopyBusyToFreeMTB THEN
bFBReset[4] := TRUE;
END_IF

IF bCopyBusyToFreeMTBRE.Q THEN
	bFBEn[4] := TRUE;
	bFBReset[4] := FALSE;
	diSinceCopyRunningTime := 0;
END_IF



	(* Convert Busy to Free MTB with Compact and sorting*)

	fbV2SubMTBFreeSlotGenerator(
		bReset									:=			bFBReset[4] ,
		AR3SiMTBBusyArm_In						:=			AR3SiMTBBusyArm_Main ,
		AR3SiMTBBusyStn_In						:=			AR3SiMTBBusyStn_Main ,
		AR3SiMTBBusyUld_In						:=			AR3SiMTBBusyUld_Main ,
		ARiArmID								:=			ARiArmID ,
		ARiUldStnID								:=			ARiUldStnID ,
		bEn										:=			bFBEn[4] ,
		AR3SiSortedMTBFreeArm_Out				:=			AR3SiSortedMTBFreeArm_Out ,
		AR3SiSortedMTBFreeStn_Out				:=			AR3SiSortedMTBFreeStn_Out ,
		AR3SiSortedMTBFreeUld_Out				:=			AR3SiSortedMTBFreeUld_Out ,
		ARiMTBFreeSlotDataQtyArm				:=			ARiMTBFreeSlotDataQtyArm ,
		ARiMTBFreeSlotDataQtyStn				:=			ARiMTBFreeSlotDataQtyStn ,
		ARiMTBFreeSlotDataQtyUld				:=			ARiMTBFreeSlotDataQtyUld  ,
		bMTBEmpty								=>			bCopiedMTBEmptyFlag ,
		bDone									=>			bFBDone[4] );

IF bCopyBusyToFreeMTB AND bFBDone[4] THEN
bCopyDone := TRUE;
ELSE
bCopyDone := FALSE;
END_IF



(***************************************************************** MTB Write *******************************************************************************)
(*MTB Write*)
IF bWrite_RTBtoMTBRE.Q THEN
iWriteStep := 1;
END_IF

CASE iWriteStep OF

0:
bWriteBusy := FALSE;
bWriteDone := FALSE;
bWriteMTBArmBlockFullError := FALSE;
bWriteMTBStnBlockFullError := FALSE;
bWriteMTBUldBlockFullError := FALSE;



1: (*Generate No Call Arm Time*)
bWriteBusy := TRUE;
bWriteMTBArmBlockFullError := FALSE;
bWriteMTBStnBlockFullError := FALSE;
bWriteMTBUldBlockFullError := FALSE;

bFBEn[1] := TRUE;
fbV2SubRTBGenerateNoCallArmTime(
	bReset									:=bFBReset[1]		,
	iLoadingCallArmTime						:=iLoadingCallArmTime		,
	AR2SiRecipeTimeBlockWithCallArmTime		:=AR2SiRecipeTimeBlockWithCallArmTime		,
	bEn										:=bFBEn[1]		,
	bDone									=>bFBDone[1]		,
	AR2SiRecipeTimeBlockNoCallArmTime		=>AR2SiRecipeTimeBlockNoCallArmTime		);

IF bFBDone[1] THEN
iWriteStep := 2;
bFBEn[1] := FALSE;
END_IF


2: (*Check RTB Block Qty - End Step*)

bFBEn[2] := TRUE;
iRTBEndStep := 0;

fbV2SubRTBEndStepFinder(
	bReset								:= bFBReset[2] ,
	AR2SiRecipeTimeBlock				:= AR2SiRecipeTimeBlockNoCallArmTime ,
	bEn									:= bFBEn[2],
	iRTB_EndStep						:= iRTBEndStep,
	bDone								=> bFBDone[2]);

IF bFBDone[2] THEN
iWriteStep := 3;
bFBEn[2] := FALSE;
END_IF

3: (*Write RTB into MTB*)
bFBEn[3] := TRUE;


	iWriteMFL := 1;
	FOR iWriteMFL := 1 TO iRTBEndStep DO
		IF iWriteMFL >= 1 AND iWriteMFL <= iRTBEndStep THEN
			iWriteSFL := 1;
			bWriteArmDone := FALSE;
			bWriteStnDone := FALSE;
			bWriteUldDone := FALSE;

			(*Check Stn types*)
			fbV2SubRTBStnTypeAltIDFinder(
				bReset									:=bFBReset[3] ,
				ARbAlternateStnEn						:=ARbAlternateStnEn ,
				AR2siAlternateStn							:=AR2siAlternateStn ,
				ARiArmID								:=ARiArmID ,
				ARiUldStnID								:=ARiUldStnID ,
				iRTBScanBlockNo						:=iWriteMFL ,
				AR2SiRecipeTimeBlock					:=AR2SiRecipeTimeBlockNoCallArmTime ,
				bEn										:=bFBEn[3] ,
				bEmptyBlockFound						=> bRTBEmptyBlockFound ,
				bArmIDFound								=> bRTBArmIDFound ,
				bStnIDFound								=> bRTBStnIDFound,
				bUldIDFound								=> bRTBUldIDFound,
				bAltStnIDFound							=> bRTBAltStnIDFound,
				iArmAdd									=> iRTBArmAdd,
				iStnAdd									=> iRTBStnAdd,
				iUldAdd									=> iRTBUldAdd,
				ARiAltStnIDFound							=> ARiRTBAltStnIDFound ,
				ARiAltStnAddFound						=> ARiRTBAltStnAddFound ,
				bDone									=> bFBDone[3]);


			(*Write Start*)
			IF (bRTBArmIDFound OR bRTBStnIDFound OR bRTBUldIDFound) AND iWriteSFL>=1 AND iWriteSFL <= iMasterBlockQty THEN

				FOR iWriteSFL := 1 TO iMasterBlockQty DO

					(*Arm Scanning*)
					IF bRTBArmIDFound THEN

						IF AR3SiMTBBusyArm_Main[iRTBArmAdd,iWriteSFL, 2] = 0 THEN

						AR3SiMTBBusyArm_Main[iRTBArmAdd,iWriteSFL, 1] := AR2SiRecipeTimeBlockNoCallArmTime[iWriteMFL, 1];
						AR3SiMTBBusyArm_Main[iRTBArmAdd,iWriteSFL, 2] := AR2SiRecipeTimeBlockNoCallArmTime[iWriteMFL, 2];
						AR3SiMTBBusyArm_Main[iRTBArmAdd,iWriteSFL, 3] := AR2SiRecipeTimeBlockNoCallArmTime[iWriteMFL, 3];
						bWriteArmDone := TRUE;
						iWriteSFL:=iMasterBlockQty+1;
						END_IF

					END_IF

					(*Stn Scanning*)
					IF bRTBStnIDFound THEN

						IF AR3SiMTBBusyStn_Main[iRTBStnAdd,iWriteSFL, 2] = 0 THEN

						AR3SiMTBBusyStn_Main[iRTBStnAdd,iWriteSFL, 1] := AR2SiRecipeTimeBlockNoCallArmTime[iWriteMFL, 1];
						AR3SiMTBBusyStn_Main[iRTBStnAdd,iWriteSFL, 2] := AR2SiRecipeTimeBlockNoCallArmTime[iWriteMFL, 2];
						AR3SiMTBBusyStn_Main[iRTBStnAdd,iWriteSFL, 3] := AR2SiRecipeTimeBlockNoCallArmTime[iWriteMFL, 3];
						bWriteStnDone := TRUE;
						iWriteSFL:=iMasterBlockQty+1;
						END_IF

					END_IF


					(*Uld Scanning*)
					IF bRTBUldIDFound THEN

						IF AR3SiMTBBusyUld_Main[iRTBUldAdd,iWriteSFL, 2] = 0 THEN

						AR3SiMTBBusyUld_Main[iRTBUldAdd,iWriteSFL, 1] := AR2SiRecipeTimeBlockNoCallArmTime[iWriteMFL, 1];
						AR3SiMTBBusyUld_Main[iRTBUldAdd,iWriteSFL, 2] := AR2SiRecipeTimeBlockNoCallArmTime[iWriteMFL, 2];
						AR3SiMTBBusyUld_Main[iRTBUldAdd,iWriteSFL, 3] := AR2SiRecipeTimeBlockNoCallArmTime[iWriteMFL, 3];
						bWriteUldDone := TRUE;
						iWriteSFL:=iMasterBlockQty+1;
						END_IF

					END_IF

				END_FOR




				IF iWriteSFL > iMasterBlockQty AND bRTBArmIDFound AND NOT bWriteArmDone THEN
				iWriteStep := 21;  (*Error!!! No Space for Arm data to fill*)
				END_IF

				IF iWriteSFL > iMasterBlockQty AND bRTBStnIDFound AND NOT bWriteStnDone THEN
				iWriteStep := 22;  (*Error!!! No Space for Stn data to fill*)
				END_IF

				IF iWriteSFL > iMasterBlockQty AND bRTBUldIDFound AND NOT bWriteUldDone THEN
				iWriteStep := 23;  (*Error!!! No Space for Uld data to fill*)
				END_IF

			END_IF

		END_IF

	END_FOR


IF iWriteMFL > iRTBEndStep AND iWriteSFL > iMasterBlockQty THEN
iWriteStep := 4;
bWriteDone := TRUE;
END_IF


4: (*Write Done Indicator*)
IF tWriteDoneTimer.Q THEN
iWriteStep := 0;
END_IF


21:; (*Error!!! No Space for Arm data to fill*)
bWriteMTBArmBlockFullError := TRUE;

22:; (*Error!!! No Space for Stn data to fill*)
bWriteMTBStnBlockFullError := TRUE;

23:; (*Error!!! No Space for Uld data to fill*)
bWriteMTBUldBlockFullError := TRUE;


END_CASE

END_FUNCTION_BLOCK

// ---- FBs/B_JKS_NewFB_V2/FBP-MTBSubFB/fbV2_SubRTBGenerateNoCallArmTime.TcPOU
FUNCTION_BLOCK fbV2_SubRTBGenerateNoCallArmTime
VAR_INPUT
	bReset			: BOOL;
	iLoadingCallArmTime : INT;

	AR2SiRecipeTimeBlockWithCallArmTime 			: ARRAY[1..iRecipeBlockQty, 1..9] OF INT;

(* RecipeTimeBlockDetail
	1 - Start Time
	2 - End Time
	3 - Stn ID
	4 - Step No (Based on Product Recipe PnP Step No)
	5 - Busy Time <Duration> = EndTime - StartTime + 1; 
	6 - Min Time (Define by User -> Process Time Per Station)
	7 - Max Time (Define by User -> For Process Tank only)
	8 - Eff Time (Final Process Time, Used on Station Timer and Call Arm Used)
	9 - BusyLink Reference 
		0		=Non
		11-19 	= BusyLinkGroupMaster No 1
		21-29 	= BusyLinkGroupMaster No 2
		=================================
		91-99 	= BusyLinkGroupMaster No 9

		111-119 	= BusyLinkGroupMaster No 1 - 1st Stn ID
		121-129 	= BusyLinkGroupMaster No 1 - 2nd Stn ID
		131-139 	= BusyLinkGroupMaster No 1 - 3rd Stn ID

		211-219 	= BusyLinkGroupMaster No 2 - 1st Stn ID
		221-229 	= BusyLinkGroupMaster No 2 - 2nd Stn ID
		231-239 	= BusyLinkGroupMaster No 2 - 3rd Stn ID

		911-919 	= BusyLinkGroupMaster No 9 - 1st Stn ID
		921-929 	= BusyLinkGroupMaster No 9 - 2nd Stn ID
		931-939 	= BusyLinkGroupMaster No 9 - 3rd Stn ID

		

*)

END_VAR

VAR_IN_OUT
	bEn				: BOOL;


END_VAR



VAR_OUTPUT
	bDone : BOOL;
	AR2SiRecipeTimeBlockNoCallArmTime 			: ARRAY[1..iRecipeBlockQty, 1..9] OF INT;

END_VAR

VAR
	bResetRE: R_TRIG;
	iStep: INT;

	iRecipeCheckFL: INT;
	AR2SiRecipeTimeBlockNoCallArmTimeEmpty 			: ARRAY[1..iRecipeBlockQty, 1..9] OF INT;
END_VAR

VAR_INPUT



END_VAR


VAR PERSISTENT


END_VAR

bResetRE(CLK:=bReset , Q=> );

IF bResetRE.Q THEN
bDone := FALSE;
END_IF


IF NOT bReset AND bEn THEN

	bDone := FALSE;
	AR2SiRecipeTimeBlockNoCallArmTime := AR2SiRecipeTimeBlockNoCallArmTimeEmpty;
(*
CASE iStep OF

1:
*)
	iRecipeCheckFL := 1;
	IF iRecipeCheckFL>0 AND iRecipeCheckFL <= iRecipeBlockQty THEN
		FOR iRecipeCheckFL := 1 TO iRecipeBlockQty DO

			IF (iRecipeCheckFL = 1 OR iRecipeCheckFL = 2) AND AR2SiRecipeTimeBlockWithCallArmTime[iRecipeCheckFL,3] > 0 THEN

				AR2SiRecipeTimeBlockNoCallArmTime[iRecipeCheckFL,1] := AR2SiRecipeTimeBlockWithCallArmTime[iRecipeCheckFL,1];
				AR2SiRecipeTimeBlockNoCallArmTime[iRecipeCheckFL,2] := AR2SiRecipeTimeBlockWithCallArmTime[iRecipeCheckFL,2]-iLoadingCallArmTime;
				AR2SiRecipeTimeBlockNoCallArmTime[iRecipeCheckFL,3] := AR2SiRecipeTimeBlockWithCallArmTime[iRecipeCheckFL,3];
				AR2SiRecipeTimeBlockNoCallArmTime[iRecipeCheckFL,4] := AR2SiRecipeTimeBlockWithCallArmTime[iRecipeCheckFL,4];
				AR2SiRecipeTimeBlockNoCallArmTime[iRecipeCheckFL,5] := AR2SiRecipeTimeBlockWithCallArmTime[iRecipeCheckFL,5]-iLoadingCallArmTime;
				AR2SiRecipeTimeBlockNoCallArmTime[iRecipeCheckFL,6] := AR2SiRecipeTimeBlockWithCallArmTime[iRecipeCheckFL,6];
				AR2SiRecipeTimeBlockNoCallArmTime[iRecipeCheckFL,7] := AR2SiRecipeTimeBlockWithCallArmTime[iRecipeCheckFL,7];
				AR2SiRecipeTimeBlockNoCallArmTime[iRecipeCheckFL,8] := AR2SiRecipeTimeBlockWithCallArmTime[iRecipeCheckFL,8];
				AR2SiRecipeTimeBlockNoCallArmTime[iRecipeCheckFL,9] := AR2SiRecipeTimeBlockWithCallArmTime[iRecipeCheckFL,9];

			ELSIF iRecipeCheckFL > 1 AND AR2SiRecipeTimeBlockWithCallArmTime[iRecipeCheckFL,3] > 0 THEN

				AR2SiRecipeTimeBlockNoCallArmTime[iRecipeCheckFL,1] := AR2SiRecipeTimeBlockWithCallArmTime[iRecipeCheckFL,1]-iLoadingCallArmTime;
				AR2SiRecipeTimeBlockNoCallArmTime[iRecipeCheckFL,2] := AR2SiRecipeTimeBlockWithCallArmTime[iRecipeCheckFL,2]-iLoadingCallArmTime;
				AR2SiRecipeTimeBlockNoCallArmTime[iRecipeCheckFL,3] := AR2SiRecipeTimeBlockWithCallArmTime[iRecipeCheckFL,3];
				AR2SiRecipeTimeBlockNoCallArmTime[iRecipeCheckFL,4] := AR2SiRecipeTimeBlockWithCallArmTime[iRecipeCheckFL,4];
				AR2SiRecipeTimeBlockNoCallArmTime[iRecipeCheckFL,5] := AR2SiRecipeTimeBlockWithCallArmTime[iRecipeCheckFL,5];
				AR2SiRecipeTimeBlockNoCallArmTime[iRecipeCheckFL,6] := AR2SiRecipeTimeBlockWithCallArmTime[iRecipeCheckFL,6];
				AR2SiRecipeTimeBlockNoCallArmTime[iRecipeCheckFL,7] := AR2SiRecipeTimeBlockWithCallArmTime[iRecipeCheckFL,7];
				AR2SiRecipeTimeBlockNoCallArmTime[iRecipeCheckFL,8] := AR2SiRecipeTimeBlockWithCallArmTime[iRecipeCheckFL,8];
				AR2SiRecipeTimeBlockNoCallArmTime[iRecipeCheckFL,9] := AR2SiRecipeTimeBlockWithCallArmTime[iRecipeCheckFL,9];
			END_IF
		END_FOR
	END_IF


bDone := TRUE;
bEn := FALSE;

(*
iStep := 12;
3:;

END_CASE
*)

END_IF

END_FUNCTION_BLOCK

// ---- FBs/B_JKS_NewFB_V2/FBP-MTBSubFB/fbV2_SubRTBEndStepFinder.TcPOU
FUNCTION_BLOCK fbV2_SubRTBEndStepFinder
VAR_INPUT
	bReset			: BOOL;
	AR2SiRecipeTimeBlock 			: ARRAY[1..iRecipeBlockQty, 1..9] OF INT;


END_VAR

VAR_IN_OUT
	bEn				: BOOL;
	iRTB_EndStep					: INT;


END_VAR



VAR_OUTPUT
	bDone : BOOL;
END_VAR

VAR
	bResetRE: R_TRIG;

	iRtbFL: INT;
END_VAR

VAR_INPUT


(* RecipeTimeBlockDetail
	1 - Start Time
	2 - End Time
	3 - Stn ID
	4 - Step No (Based on Product Recipe PnP Step No)
	5 - Busy Time <Duration> = EndTime - StartTime + 1; 
	6 - Min Time (Define by User -> Process Time Per Station)
	7 - Max Time (Define by User -> For Process Tank only)
	8 - Eff Time (Final Process Time, Used on Station Timer and Call Arm Used)
	9 - BusyLink Reference ( 0=Non, 1~9=BusyLinkGroupMaster No, 11-19=Group1Slave, 21-29=Group2Slave ~ 91-99=Group9Slave)
*)

END_VAR


VAR PERSISTENT


END_VAR

bResetRE(CLK:=bReset , Q=> );

IF bResetRE.Q THEN
iRTB_EndStep := 0;
bDone := FALSE;
END_IF

(*
IF NOT bEn THEN
bDone := FALSE;
END_IF
*)


IF NOT bReset AND bEn THEN
bDone := FALSE;
iRTB_EndStep := 0;
	iRtbFL := 1;
	FOR iRtbFL := 1 TO iRecipeBlockQty DO
		IF iRtbFL >= 1 AND iRtbFL <= iRecipeBlockQty THEN
			IF AR2SiRecipeTimeBlock[iRtbFL , 3] > 0 THEN
			iRTB_EndStep := iRtbFL;
			END_IF
		END_IF
	END_FOR

bDone := TRUE;
bEn := FALSE;
END_IF

END_FUNCTION_BLOCK

// ---- FBs/B_JKS_NewFB_V2/FBP-MTBSubFB/fbV2_SubRTBStnTypeAltIDFinder.TcPOU
FUNCTION_BLOCK fbV2_SubRTBStnTypeAltIDFinder
VAR_INPUT
	bReset																		: BOOL;
	ARbAlternateStnEn 															: ARRAY [1..iAlternateSetQty] OF BOOL;
	AR2siAlternateStn 																: ARRAY [1..iAlternateSetQty, 1..iAlternateStnQty] OF INT;
	ARiArmID																	: ARRAY [1..iArmQty] OF INT;
	ARiUldStnID																	: ARRAY [1..iUldStnQty] OF INT;		(* To Define Unloading Station ID*)

	iRTBScanBlockNo															: INT;
	AR2SiRecipeTimeBlock				 										: ARRAY[1..iRecipeBlockQty, 1..9] OF INT;

(* RecipeTimeBlockDetail
	1 - Start Time
	2 - End Time
	3 - Stn ID
	4 - Step No (Based on Product Recipe PnP Step No)
	5 - Busy Time <Duration> = EndTime - StartTime + 1; 
	6 - Min Time (Define by User -> Process Time Per Station)
	7 - Max Time (Define by User -> For Process Tank only)
	8 - Eff Time (Final Process Time, Used on Station Timer and Call Arm Used)
	9 - BusyLink Reference 
		0		=Non
		11-19 	= BusyLinkGroupMaster No 1
		21-29 	= BusyLinkGroupMaster No 2
		=================================
		91-99 	= BusyLinkGroupMaster No 9

		111-119 	= BusyLinkGroupMaster No 1 - 1st Stn ID
		121-129 	= BusyLinkGroupMaster No 1 - 2nd Stn ID
		131-139 	= BusyLinkGroupMaster No 1 - 3rd Stn ID

		211-219 	= BusyLinkGroupMaster No 2 - 1st Stn ID
		221-229 	= BusyLinkGroupMaster No 2 - 2nd Stn ID
		231-239 	= BusyLinkGroupMaster No 2 - 3rd Stn ID

		911-919 	= BusyLinkGroupMaster No 9 - 1st Stn ID
		921-929 	= BusyLinkGroupMaster No 9 - 2nd Stn ID
		931-939 	= BusyLinkGroupMaster No 9 - 3rd Stn ID

		

*)

END_VAR

VAR_IN_OUT
	bEn										: BOOL;


END_VAR



VAR_OUTPUT
	bEmptyBlockFound						: BOOL;
	bArmIDFound								: BOOL;
	bStnIDFound								: BOOL;
	bUldIDFound								: BOOL;
	bAltStnIDFound							: BOOL;
	iArmAdd									: INT;
	iStnAdd									: INT;
	iUldAdd									: INT;
	ARiAltStnIDFound							: ARRAY [1..iAlternateStnQty] OF INT;
	ARiAltStnAddFound						: ARRAY [1..iAlternateStnQty] OF INT;
	bDone : BOOL;
END_VAR

VAR
	bResetRE					: R_TRIG;

	iCheckAlternateStnEnFL 		: INT;
	iClearBufferAltFL 				: INT;
	iCheckArmIDFL 				: INT;
	iCheckStnIDFL 				: INT;
	iCheckUldIDFL 				: INT;
	iAlternateSetFindFL 			: INT;
	iAlternateStnFindFL 			: INT;
	iAltStnTransferFL 				: INT;
	iAltStnAddCheckFL 			: INT;
	iAltStnAddCheckSFL 			: INT;


	bAlternateStnEnableFound 		: BOOL;
	ARiAltStnIDFoundEmpty		: ARRAY [1..iAlternateStnQty] OF INT;
	ARiAltStnAddFoundEmpty		: ARRAY [1..iAlternateStnQty] OF INT;
	iRTBScanBlockNoPrevious: INT;
	bEnFE: F_TRIG;
	bEnRE: R_TRIG;
END_VAR



VAR PERSISTENT


END_VAR

bResetRE(CLK:=bReset , Q=> );
bEnFE(CLK:=bEn , Q=> );
bEnRE(CLK:=bEn , Q=> );

IF bResetRE.Q OR bEnFE.Q THEN

	bEn						:= FALSE;
	bDone 					:= FALSE;

	bEmptyBlockFound		:= FALSE;
	bArmIDFound	 			:= FALSE;
	bStnIDFound 				:= FALSE;
	bUldIDFound	 			:= FALSE;
	bAltStnIDFound			:= FALSE;
	iArmAdd 					:= 0;
	iStnAdd 					:= 0;
	iUldAdd 					:= 0;
	ARiAltStnIDFound			:= ARiAltStnIDFoundEmpty;
	ARiAltStnAddFound		:= ARiAltStnAddFoundEmpty;

	bAlternateStnEnableFound 	:= FALSE;
	iRTBScanBlockNoPrevious := iRTBScanBlockNo;


END_IF

(*
IF NOT bEn THEN
bDone := FALSE;
END_IF
*)


IF
NOT bReset
AND bEn
AND (iRTBScanBlockNoPrevious <> iRTBScanBlockNo OR bEnRE.Q)
THEN
	bDone 					:= FALSE;

	bEmptyBlockFound		:= FALSE;
	bArmIDFound	 			:= FALSE;
	bStnIDFound 				:= FALSE;
	bUldIDFound	 			:= FALSE;
	bAltStnIDFound			:= FALSE;
	iArmAdd 					:= 0;
	iStnAdd 					:= 0;
	iUldAdd 					:= 0;
	ARiAltStnIDFound			:= ARiAltStnIDFoundEmpty;
	ARiAltStnAddFound		:= ARiAltStnAddFoundEmpty;

	bAlternateStnEnableFound 	:= FALSE;

	IF AR2SiRecipeTimeBlock[iRTBScanBlockNo,3] > 0
	AND iRTBScanBlockNo > 0 AND iRTBScanBlockNo <= iRecipeBlockQty
	THEN
	
		(*Check if AlternateStn Enable*)
		iCheckAlternateStnEnFL := 1;
		FOR iCheckAlternateStnEnFL := 1 TO iAlternateSetQty DO
			IF iCheckAlternateStnEnFL >= 1 AND iCheckAlternateStnEnFL <= iAlternateSetQty THEN
				IF ARbAlternateStnEn[iCheckAlternateStnEnFL] THEN
					bAlternateStnEnableFound := TRUE;
				END_IF
			END_IF
		END_FOR
	


	
		(*Check ArmID*)
		iCheckArmIDFL := 1;
		IF iCheckArmIDFL>0 AND iCheckArmIDFL < iArmQty+1 THEN
			FOR iCheckArmIDFL := 1 TO iArmQty DO
				IF AR2SiRecipeTimeBlock[iRTBScanBlockNo,3] = ARiArmID[iCheckArmIDFL] THEN
				iArmAdd := iCheckArmIDFL;
				bArmIDFound := TRUE;
				iCheckArmIDFL := iArmQty+1;
				END_IF
			END_FOR
		END_IF

		(*Check StnID*)
		iCheckStnIDFL := 1;
		IF iCheckStnIDFL>0 AND iCheckStnIDFL <iStnQty+1 THEN
			FOR iCheckStnIDFL := 1 TO iStnQty DO
				IF AR2SiRecipeTimeBlock[iRTBScanBlockNo,3] = iCheckStnIDFL THEN
				iStnAdd := iCheckStnIDFL;
				bStnIDFound := TRUE;
				iCheckStnIDFL := iStnQty+1;
				END_IF
			END_FOR
		END_IF

		(*Check UldID*)
		iCheckUldIDFL := 1;
		IF iCheckUldIDFL>0 AND iCheckUldIDFL <iUldStnQty+1 THEN
			FOR iCheckUldIDFL := 1 TO iUldStnQty DO
				IF AR2SiRecipeTimeBlock[iRTBScanBlockNo,3] = ARiUldStnID[iCheckUldIDFL] THEN
				iUldAdd := iCheckUldIDFL;
				bUldIDFound := TRUE;
				iCheckUldIDFL := iUldStnQty+1;
				END_IF
			END_FOR
		END_IF
	
		IF (bStnIDFound OR bUldIDFound) AND bAlternateStnEnableFound THEN
		iAlternateSetFindFL := 1;
			FOR iAlternateSetFindFL := 1 TO iAlternateSetQty DO
				IF iAlternateSetFindFL >= 1 AND iAlternateSetFindFL <= iAlternateSetQty THEN
					IF ARbAlternateStnEn[iAlternateSetFindFL] THEN
					iAlternateStnFindFL := 1; (*Find Stn ID matching*)
						FOR iAlternateStnFindFL := 1 TO iAlternateStnQty DO
							IF iAlternateStnFindFL >= 1 AND iAlternateStnFindFL <= iAlternateStnQty THEN
								IF (bStnIDFound AND iStnAdd = AR2SiAlternateStn[iAlternateSetFindFL , iAlternateStnFindFL])
								OR (bUldIDFound AND ARiUldStnID[iUldAdd] = AR2SiAlternateStn[iAlternateSetFindFL , iAlternateStnFindFL])
								 THEN
									bAltStnIDFound := TRUE;
									iAltStnTransferFL := 1;
	
										FOR iAltStnTransferFL := 1 TO iAlternateStnQty DO
											IF iAltStnTransferFL >= 1 AND iAltStnTransferFL <= iAlternateStnQty THEN
												ARiAltStnIDFound[iAltStnTransferFL] := AR2SiAlternateStn[iAlternateSetFindFL , iAltStnTransferFL];
											END_IF
										END_FOR
	
	
									iAltStnAddCheckFL := 1;
	
										FOR iAltStnAddCheckFL := 1 TO iAlternateStnQty DO
											IF iAltStnAddCheckFL >= 1 AND iAltStnAddCheckFL <= iAlternateStnQty THEN
												IF (*bStnIDFound*)ARiAltStnIDFound[iAltStnAddCheckFL] >= 1 AND ARiAltStnIDFound[iAltStnAddCheckFL] <= iStnQty THEN
	
													ARiAltStnAddFound[iAltStnAddCheckFL] := ARiAltStnIDFound[iAltStnAddCheckFL];
	
												ELSIF (*bUldIDFound*) ARiAltStnIDFound[iAltStnAddCheckFL] > 0 THEN
												iAltStnAddCheckSFL := 1;
													FOR iAltStnAddCheckSFL := 1 TO iUldStnQty DO
														IF iAltStnAddCheckSFL >= 1 AND iAltStnAddCheckSFL <= iUldStnQty THEN
															IF ARiAltStnIDFound[iAltStnAddCheckFL] = ARiUldStnID[iAltStnAddCheckSFL] THEN
															ARiAltStnAddFound[iAltStnAddCheckFL] := iAltStnAddCheckSFL;
															END_IF
														END_IF
	
													END_FOR
												ELSE
	
													ARiAltStnAddFound[iAltStnAddCheckFL] := 0;
	

												END_IF
	
											END_IF
										END_FOR
	
	
									iAlternateSetFindFL := iAlternateSetQty+1;
									iAlternateStnFindFL := iAlternateStnQty+1;
									iAltStnTransferFL := iAlternateStnQty+1;
	
								END_IF
							END_IF
						END_FOR
					END_IF
				END_IF
			END_FOR
		END_IF

	bDone 						:= TRUE;
	iRTBScanBlockNoPrevious 	:= iRTBScanBlockNo;
	ELSE
	bEmptyBlockFound			:= TRUE;
	bDone 						:= TRUE;
	iRTBScanBlockNoPrevious 	:= iRTBScanBlockNo;
	END_IF

ELSE
iRTBScanBlockNoPrevious := iRTBScanBlockNo;
END_IF

END_FUNCTION_BLOCK

// ---- FBs/B_JKS_NewFB_V2/FBP-MTBSubFB/fbV2_SubRTBBusyLinkMTSUpdate.TcPOU
FUNCTION_BLOCK fbV2_SubRTBBusyLinkMTSUpdate
VAR_INPUT
	bReset			: BOOL;


END_VAR

VAR_IN_OUT
	bEn				: BOOL;
	AR2SiRecipeTimeBlockWithCallArmTime 			: ARRAY[1..iRecipeBlockQty, 1..9] OF INT;

(* RecipeTimeBlockDetail
	1 - Start Time
	2 - End Time
	3 - Stn ID
	4 - Step No (Based on Product Recipe PnP Step No)
	5 - Busy Time <Duration> = EndTime - StartTime + 1; 
	6 - Min Time (Define by User -> Process Time Per Station)
	7 - Max Time (Define by User -> For Process Tank only)
	8 - Eff Time (Final Process Time, Used on Station Timer and Call Arm Used)
	9 - BusyLink Reference 
		0		=Non
		11-19 	= BusyLinkGroupMaster No 1
		21-29 	= BusyLinkGroupMaster No 2
		=================================
		91-99 	= BusyLinkGroupMaster No 9

		111-119 	= BusyLinkGroupMaster No 1 - 1st Stn ID
		121-129 	= BusyLinkGroupMaster No 1 - 2nd Stn ID
		131-139 	= BusyLinkGroupMaster No 1 - 3rd Stn ID

		211-219 	= BusyLinkGroupMaster No 2 - 1st Stn ID
		221-229 	= BusyLinkGroupMaster No 2 - 2nd Stn ID
		231-239 	= BusyLinkGroupMaster No 2 - 3rd Stn ID

		911-919 	= BusyLinkGroupMaster No 9 - 1st Stn ID
		921-929 	= BusyLinkGroupMaster No 9 - 2nd Stn ID
		931-939 	= BusyLinkGroupMaster No 9 - 3rd Stn ID

		

*)

END_VAR



VAR_OUTPUT
	bDone : BOOL;
END_VAR

VAR
	bResetRE: R_TRIG;
	iStep: INT;

	iRtbFL: INT;
	iBufferBusyLinkGroup : ARRAY[1..iBusyLinkUpSetQty(*5*),1..iBusyLinkUpStnQty(*6*), 1..9] OF INT; (* 9 Groups Max*)
	iBusySetFL: INT;
	iBusyStnFL: INT;
	iRecipeCheckFL: INT;
END_VAR

VAR_INPUT


(* RecipeTimeBlockDetail
	1 - Start Time
	2 - End Time
	3 - Stn ID
	4 - Step No (Based on Product Recipe PnP Step No)
	5 - Busy Time <Duration> = EndTime - StartTime + 1; 
	6 - Min Time (Define by User -> Process Time Per Station)
	7 - Max Time (Define by User -> For Process Tank only)
	8 - Eff Time (Final Process Time, Used on Station Timer and Call Arm Used)
	9 - BusyLink Reference ( 0=Non, 1~9=BusyLinkGroupMaster No, 11-19=Group1Slave, 21-29=Group2Slave ~ 91-99=Group9Slave)
*)

END_VAR


VAR PERSISTENT


END_VAR

bResetRE(CLK:=bReset , Q=> );

IF bResetRE.Q THEN
bDone := FALSE;
END_IF

(*
IF NOT bEn THEN
bDone := FALSE;
END_IF
*)


IF NOT bReset AND bEn THEN
bDone := FALSE;
(*
CASE iStep OF

1:
*)
	iRecipeCheckFL := 1;
	IF iRecipeCheckFL>0 AND iRecipeCheckFL <= iRecipeBlockQty THEN
		FOR iRecipeCheckFL := 1 TO iRecipeBlockQty DO

			iBusySetFL := 1;
			IF iBusySetFL>= 1 AND iBusySetFL <= iBusyLinkUpSetQty THEN
				FOR iBusySetFL := 1 TO iBusyLinkUpSetQty DO


					iBusyStnFL := 1;
					IF iBusyStnFL>= 1 AND iBusyStnFL <= iBusyLinkUpStnQty THEN
						FOR iBusyStnFL := 1 TO iBusyLinkUpStnQty DO
							IF AR2SiRecipeTimeBlockWithCallArmTime[iRecipeCheckFL,9] = (iBusySetFL*10)+iBusyStnFL THEN
		
								iBufferBusyLinkGroup[iBusySetFL, iBusyStnFL,1] := AR2SiRecipeTimeBlockWithCallArmTime[iRecipeCheckFL,1];
								iBufferBusyLinkGroup[iBusySetFL, iBusyStnFL,2] := AR2SiRecipeTimeBlockWithCallArmTime[iRecipeCheckFL,2];
								iBufferBusyLinkGroup[iBusySetFL, iBusyStnFL,3] := AR2SiRecipeTimeBlockWithCallArmTime[iRecipeCheckFL,3];
								iBufferBusyLinkGroup[iBusySetFL, iBusyStnFL,4] := AR2SiRecipeTimeBlockWithCallArmTime[iRecipeCheckFL,4];
								iBufferBusyLinkGroup[iBusySetFL, iBusyStnFL,5] := AR2SiRecipeTimeBlockWithCallArmTime[iRecipeCheckFL,5];
								iBufferBusyLinkGroup[iBusySetFL, iBusyStnFL,6] := AR2SiRecipeTimeBlockWithCallArmTime[iRecipeCheckFL,6];
								iBufferBusyLinkGroup[iBusySetFL, iBusyStnFL,7] := AR2SiRecipeTimeBlockWithCallArmTime[iRecipeCheckFL,7];
								iBufferBusyLinkGroup[iBusySetFL, iBusyStnFL,8] := AR2SiRecipeTimeBlockWithCallArmTime[iRecipeCheckFL,8];
								iBufferBusyLinkGroup[iBusySetFL, iBusyStnFL,9] := AR2SiRecipeTimeBlockWithCallArmTime[iRecipeCheckFL,9];
		
							END_IF
						END_FOR
					END_IF

				END_FOR
			END_IF

		END_FOR
	END_IF
(*iStep := 11;
2:
*)	iRecipeCheckFL := 1;
	IF iRecipeCheckFL>0 AND iRecipeCheckFL <= iRecipeBlockQty THEN
		FOR iRecipeCheckFL := 1 TO iRecipeBlockQty DO

			iBusySetFL := 1;
			IF iBusySetFL>= 1 AND iBusySetFL <= iBusyLinkUpSetQty THEN
				FOR iBusySetFL := 1 TO iBusyLinkUpSetQty DO

					iBusyStnFL := 1;
					IF iBusyStnFL>= 1 AND iBusyStnFL <= iBusyLinkUpStnQty THEN
						FOR iBusyStnFL := 1 TO iBusyLinkUpStnQty DO
		
							IF iBufferBusyLinkGroup[iBusySetFL, iBusyStnFL,9] > 0 THEN
								IF AR2SiRecipeTimeBlockWithCallArmTime[iRecipeCheckFL,9] > (iBufferBusyLinkGroup[iBusySetFL, iBusyStnFL,9]*10)
								AND AR2SiRecipeTimeBlockWithCallArmTime[iRecipeCheckFL,9] < ((iBufferBusyLinkGroup[iBusySetFL, iBusyStnFL,9]+1)*10) THEN
		
									AR2SiRecipeTimeBlockWithCallArmTime[iRecipeCheckFL,1] := iBufferBusyLinkGroup[iBusySetFL, iBusyStnFL,1];
									AR2SiRecipeTimeBlockWithCallArmTime[iRecipeCheckFL,2] := iBufferBusyLinkGroup[iBusySetFL, iBusyStnFL,2];
									(*AR2SiRecipeTimeBlockWithCallArmTime[iRecipeCheckFL,3] := iBufferBusyLinkGroup[iBusySetFL, iBusyStnFL,3];*)
									AR2SiRecipeTimeBlockWithCallArmTime[iRecipeCheckFL,4] := iBufferBusyLinkGroup[iBusySetFL, iBusyStnFL,4];
									AR2SiRecipeTimeBlockWithCallArmTime[iRecipeCheckFL,5] := iBufferBusyLinkGroup[iBusySetFL, iBusyStnFL,5];
									AR2SiRecipeTimeBlockWithCallArmTime[iRecipeCheckFL,6] := iBufferBusyLinkGroup[iBusySetFL, iBusyStnFL,6];
									AR2SiRecipeTimeBlockWithCallArmTime[iRecipeCheckFL,7] := iBufferBusyLinkGroup[iBusySetFL, iBusyStnFL,7];
									AR2SiRecipeTimeBlockWithCallArmTime[iRecipeCheckFL,8] := iBufferBusyLinkGroup[iBusySetFL, iBusyStnFL,8];
									(*AR2SiRecipeTimeBlockWithCallArmTime[iRecipeCheckFL,9] := iBufferBusyLinkGroup[iBusySetFL, iBusyStnFL,9];*)
		
								END_IF
							END_IF

						END_FOR
					END_IF
				END_FOR
			END_IF
		END_FOR
	END_IF


bDone := TRUE;
bEn := FALSE;

(*
iStep := 12;
3:;

END_CASE
*)

END_IF

END_FUNCTION_BLOCK

// ---- FBs/B_JKS_NewFB_V2/FBP-MTBSubFB/fbV2_SubTimeBlockCompare.TcPOU
FUNCTION_BLOCK fbV2_SubTimeBlockCompare
VAR_INPUT
	bEn				: BOOL;
	iMasterDataStart : INT;
	iMasterDataEnd : INT;
	iRecipeDataStart : INT;
	iRecipeDataEnd : INT;
END_VAR
VAR_IN_OUT
	bSourceDataError: BOOL;
	bCrashFound : BOOL;
	bNoCrashFound: BOOL;
	iShiftValue : INT;

END_VAR
VAR

	bEnFE: F_TRIG;
END_VAR

bEnFE(CLK:=bEn , Q=> );

IF bEnFE.Q THEN

	bSourceDataError := FALSE;
	bCrashFound := FALSE;
	bNoCrashFound := FALSE;
	iShiftValue := 0;

END_IF


IF bEn THEN
	IF iMasterDataStart (*MD1*)  >= 0 AND  iMasterDataEnd (*MD2*)  >= 1 AND iRecipeDataStart (*RD1*)  >= 0 AND  iRecipeDataEnd (*RD2*)  >= 1AND iMasterDataStart (*MD1*)  < iMasterDataEnd (*MD2*)  AND iRecipeDataStart (*RD1*)  < iRecipeDataEnd (*RD2*)  THEN
	
	
		IF 	(iMasterDataStart (*MD1*)  <= iRecipeDataStart (*RD1*)  AND iMasterDataEnd (*MD2*)  >= iRecipeDataStart (*RD1*) )
		OR 	(iMasterDataStart (*MD1*)  <= iRecipeDataEnd (*RD2*)  AND iMasterDataEnd (*MD2*)  >= iRecipeDataEnd (*RD2*) )
		OR	(iRecipeDataStart (*RD1*)  <= iMasterDataStart (*MD1*)  AND iRecipeDataEnd (*RD2*)  >= iMasterDataStart (*MD1*) )
		OR 	(iRecipeDataStart (*RD1*)  <= iMasterDataEnd (*MD2*)  AND iRecipeDataEnd (*RD2*)  >= iMasterDataEnd (*MD2*) ) THEN
		bSourceDataError := FALSE;
		bCrashFound := TRUE;
		bNoCrashFound := FALSE;
		iShiftValue := iMasterDataEnd (*MD2*)  - iRecipeDataStart (*RD1*)  +1;
		ELSE
		bSourceDataError := FALSE;
		bCrashFound := FALSE;
		bNoCrashFound := TRUE;
		iShiftValue := 0;
		END_IF


	ELSE
		bSourceDataError := TRUE;
		bCrashFound := FALSE;
		bNoCrashFound := FALSE;
		iShiftValue := 0;
	END_IF

END_IF

END_FUNCTION_BLOCK

// ---- FBs/B_JKS_NewFB_V3/XML/FB3_XmlSvrRW_MultipleGVL.TcPOU
FUNCTION_BLOCK FB3_XmlSvrRW_MultipleGVL
VAR_INPUT
	bWriteSt				: BOOL;
	bReadSt					: BOOL;
	ARp_SymAddr				: ARRAY [1..C_iXMLSrvMultiGVLQty] OF PVOID;
	ARp_SymSize				: ARRAY [1..C_iXMLSrvMultiGVLQty] OF UDINT;
	ARs_FolderName			: ARRAY [1..C_iXMLSrvMultiGVLQty] OF T_MaxString;  // Make sure the Default File Path and the Folder is Exist otherwise it will prompt Error
	ARs_VariableName		: ARRAY [1..C_iXMLSrvMultiGVLQty] OF T_MaxString;  // Make sure the Variable Name is matching with the SymAddr
	sDefaultFilePath		: STRING := 'C:\JKS\PLC\XML\';
	sFileExtension			: STRING := 'XML';
	
END_VAR
VAR_OUTPUT
	bWrite_Done				: BOOL;
	bWrite_Busy				: BOOL;
	bWrite_Error			: BOOL;
	udWrite_ErrId			: UDINT;
	bRead_Done				: BOOL;
	bRead_Busy				: BOOL;
	bRead_Error				: BOOL;
	udRead_ErrId 			: UDINT;
	iErrorArrayId			: INT;
	iTotalTime_100ms		: INT;
END_VAR

VAR
		fbXmlSrvWriteByAdd	: FB_XmlSrvWrite;
		fbXmlSrvReadByAdd	: FB_XmlSrvRead;

	bWriteStRE			: R_TRIG;
	bReadStRE			: R_TRIG;
	iArrayId			: INT;
	iFL					: INT;
	iCase				: INT;
	bFound				: BOOL;

	bWriteSt_Int		: BOOL 	:= FALSE;
	bReadSt_Int			: BOOL	:= FALSE;
	bWrite_Busy_Int		: BOOL	:= FALSE;
	bRead_Busy_Int		: BOOL	:= FALSE;
	sFilePath_Int		: T_MaxString;
	sXPath_Int			: T_MaxString;
	sFilePath_Rename	: T_MaxString;
	sFilePath_Delete	: T_MaxString;
//	bRenameSt_Int		: BOOL;
//	bRename_Busy_Int	: BOOL;
//	bDeleteSt_Int		: BOOL;
//	bDelete_Busy_Int	: BOOL;
	iSFL: INT;
	sFilenameDateToDelete: STRING;
	fbFileRename		: FB_FileRename;
	fbFileDelete		: FB_FileDelete;
	
END_VAR

IF NOT bWriteSt AND NOT bReadSt THEN
	iCase 					:= 0;

END_IF

bWriteStRE(CLK	:=bWriteSt 	, Q=> );
bReadStRE(CLK	:=bReadSt  	, Q=> );

// Capture Total Time for Read or Write
IF iCase = 1 OR (iCase >= 10 AND iCase < 19) OR (iCase >= 20 AND iCase < 29) THEN
	IF bClockPulse_0_1Sec THEN
		iTotalTime_100ms := iTotalTime_100ms + 1;
	END_IF
END_IF

IF iArrayId >= 1 THEN
	fbXmlSrvWriteByAdd(
		sNetId			:= '', 
		ePath			:= PATH_GENERIC, 
		nMode			:= XMLSRV_ADDMISSING, 
		pSymAddr		:= ARp_SymAddr[iArrayId], 
		cbSymSize		:= ARp_SymSize[iArrayId], 
		sFilePath		:= sFilePath_Int, 
		sXPath			:= sXPath_Int, 
		bExecute		:= bWriteSt_Int, 
		tTimeout		:= T#5S, 
		bBusy			=> bWrite_Busy_Int, 
		bError			=> bWrite_Error);
	
	fbXmlSrvReadByAdd(
		sNetId			:= '', 
		ePath			:= PATH_GENERIC, 
		nMode			:= XMLSRV_ADDMISSING, 
		pSymAddr		:= ARp_SymAddr[iArrayId], 
		cbSymSize		:= ARp_SymSize[iArrayId], 
		sFilePath		:= sFilePath_Int, 
		sXPath			:= sXPath_Int, 
		bExecute		:= bReadSt_Int, 
		tTimeout		:= T#5S, 
		bBusy			=> bRead_Busy_Int, 
		bError			=> bRead_Error, 
		nErrId			=> );
END_IF
	
IF 		bWriteStRE.Q 	AND NOT bReadSt 	AND NOT bRead_Busy 	THEN 	iCase := 1; 	bWrite_Busy := TRUE;
ELSIF	bReadStRE.Q		AND NOT bWriteSt 	AND NOT bWrite_Busy	THEN 	iCase := 1;		bRead_Busy := TRUE;			END_IF	


CASE iCase OF
	
	0: 	// Reset ALL

			iArrayId 				:= 0;
			iErrorArrayId			:= 0;

			udWrite_ErrId			:= 0;
			bWrite_Busy				:= FALSE;
			bWrite_Error			:= FALSE;
			bWrite_Done				:= FALSE;

			udRead_ErrId			:= 0;
			bRead_Busy				:= FALSE;
			bRead_Error				:= FALSE;
			bRead_Done				:= FALSE;

			bWriteSt_Int			:= FALSE;
			bReadSt_Int				:= FALSE;
			bWrite_Busy_Int			:= FALSE;
			bRead_Busy_Int			:= FALSE;
	
			iTotalTime_100ms		:= 0;	

			sFilePath_Int			:= '';
			sXPath_Int				:= '';	

	1: // Check Avaiable Array to trigger Read/Write

			
	
			FOR iFL := 1 TO C_iXMLSrvMultiGVLQty DO
	
				IF iArrayId+iFL <= C_iXMLSrvMultiGVLQty THEN			
					IF ARs_FolderName[iArrayId+iFL] <> '' AND ARs_VariableName[iArrayId+iFL] <> '' THEN
						iArrayId 	:= iArrayId+iFL;				
						bFound		:= TRUE;
						iFL			:= C_iXMLSrvMultiGVLQty + 1;
					END_IF
				END_IF
			END_FOR	
			
			
			IF 	bFound THEN

				sFilePath_Int	:=	concat(sDefaultFilePath,	ARs_FolderName[iArrayId]		);
				sFilePath_Int	:=	concat(sFilePath_Int,		'\'								);
				sFilePath_Int	:=	concat(sFilePath_Int,		ARs_VariableName[iArrayId]		);
				sFilePath_Int	:=	concat(sFilePath_Int,		'.'								);
				sFilePath_Int	:=	concat(sFilePath_Int,		sFileExtension					);

				sXPath_Int		:=	concat('/GVL/',				ARs_FolderName[iArrayId]		);
				sXPath_Int		:=	concat(sXPath_Int,			'/'								);
				sXPath_Int		:=	concat(sXPath_Int,			ARs_VariableName[iArrayId]		);
					
		
					IF 		bWrite_Busy THEN		
							iCase 	:= 12;					
							bFound 	:= FALSE;
					
					ELSIF 	bRead_Busy THEN		
							iCase 	:= 22;					
							bFound 	:= FALSE;
					END_IF			

			ELSE
			
					IF 		bWrite_Busy THEN	iCase	:= 19; 			// Write Done
					ELSIF	bRead_Busy 	THEN	iCase	:= 29; END_IF 	// Read Done

			END_IF	

	12: // Check Previous Write date and prepare to rename before write
	
				IF AR2sXMLMultipleGVLVerDate[iArrayId][1] = DSLocalSystemTimeML.sCurrentDate_General THEN // Same date, no shifting required, Proceed Write/Overwrite
					iCase := 17;
				ELSE

					sFilenameDateToDelete := AR2sXMLMultipleGVLVerDate[iArrayId][C_iXMLMultipleGVLVerQty];
					AR2sXMLMultipleGVLVerDate[iArrayId][C_iXMLMultipleGVLVerQty] := '';

					FOR iSFL := 1 TO C_iXMLMultipleGVLVerQty DO
						IF iSFL < C_iXMLMultipleGVLVerQty THEN
							AR2sXMLMultipleGVLVerDate[iArrayId][C_iXMLMultipleGVLVerQty-iSFL+1] := AR2sXMLMultipleGVLVerDate[iArrayId][C_iXMLMultipleGVLVerQty-iSFL];
						ELSIF iSFL = C_iXMLMultipleGVLVerQty THEN
							AR2sXMLMultipleGVLVerDate[iArrayId][1] := '';
						END_IF
					END_FOR

					IF sFilenameDateToDelete <> '' THEN
						iCase := 13; // Proceed to delete Outdated MultipleGVL XML
					ELSE
						iCase := 15; // Proceed to Rename MultipleGVL XML
					END_IF


				END_IF

				
	13: // Delete File

				sFilePath_Delete	:=	concat(sDefaultFilePath,	ARs_FolderName[iArrayId]					);
				sFilePath_Delete	:=	concat(sFilePath_Delete,	'\'											);
				sFilePath_Delete	:=	concat(sFilePath_Delete,	ARs_VariableName[iArrayId]					);
				sFilePath_Delete	:=	concat(sFilePath_Delete,	'_'											);
				sFilePath_Delete	:=	concat(sFilePath_Delete,	sFilenameDateToDelete						);
				sFilePath_Delete	:=	concat(sFilePath_Delete,	'.'											);
				sFilePath_Delete	:=	concat(sFilePath_Delete,	sFileExtension								);

			fbFileDelete(bExecute	:= FALSE);	
			fbFileDelete(
						sPathName	:= sFilePath_Delete, 
						ePath		:= PATH_GENERIC, 
						bExecute	:= TRUE);
						
			IF fbFileDelete.bBusy THEN
				iCase := 14; // Wait Delete FB to complete
			END_IF


	14: // Delete File - Verify completion
			fbFileDelete(bExecute	:= FALSE);	
			IF NOT fbFileDelete.bBusy THEN
				iCase := 15; // Proceed to rename file regardless the the said file being delete (if found) or not found
			END_IF
			
	15: // Rename File

				sFilePath_Rename	:=	concat(sDefaultFilePath,	ARs_FolderName[iArrayId]					);
				sFilePath_Rename	:=	concat(sFilePath_Rename,	'\'											);
				sFilePath_Rename	:=	concat(sFilePath_Rename,	ARs_VariableName[iArrayId]					);
				sFilePath_Rename	:=	concat(sFilePath_Rename,	'_'											);
				sFilePath_Rename	:=	concat(sFilePath_Rename,	DSLocalSystemTimeML.sCurrentDate_General	);
				sFilePath_Rename	:=	concat(sFilePath_Rename,	'.'											);
				sFilePath_Rename	:=	concat(sFilePath_Rename,	sFileExtension								);
			
			fbFileRename(bExecute	:= FALSE);	
			fbFileRename(
						sOldName		:= sFilePath_Int, 
						sNewName		:= sFilePath_Rename, 
						ePath			:= PATH_GENERIC, 
						bExecute		:= TRUE ); 
			
			IF fbFileRename.bBusy THEN
				iCase := 16; // Wait Rename FB to complete
			END_IF

	16: // Rename File - Verify completion
			fbFileRename(bExecute	:= FALSE);	
			IF NOT fbFileRename.bBusy THEN
				iCase := 17; // Proceed to Write file regardless the the said file being rename (if found) or not found
				AR2sXMLMultipleGVLVerDate[iArrayId][1] := DSLocalSystemTimeML.sCurrentDate_General;
			END_IF
						
	17: // Write Start

			bWriteSt_Int := TRUE;
	
			IF fbXmlSrvWriteByAdd.bExecute AND NOT fbXmlSrvWriteByAdd.bBusy AND NOT fbXmlSrvWriteByAdd.bError 
			AND fbXmlSrvWriteByAdd.sFilePath 	= sFilePath_Int
			AND fbXmlSrvWriteByAdd.sXPath		= sXPath_Int	THEN
				iCase := 18; // Write Done -> Proceed to clear FB to prepare for Next Cycle (Array) 			
				
			ELSIF fbXmlSrvWriteByAdd.bError THEN
				udWrite_ErrId := fbXmlSrvWriteByAdd.nErrId;
				iCase := 99;	// WRITE ERROR
				iErrorArrayId	:= iArrayId;
			END_IF

	18: 	//  Write - prepare for Next Cycle (Array) 
			
			bWriteSt_Int := FALSE;
	
			IF NOT fbXmlSrvWriteByAdd.bExecute AND NOT fbXmlSrvWriteByAdd.bBusy  THEN
				iCase := 1; // Proceed to Next Cycle (Array) 
			END_IF
		
		
	19: // Write - All Done 
		
			bWrite_Busy 	:= FALSE;
			bWrite_Done 	:= TRUE;
			
	22: // Read Start

			bReadSt_Int := TRUE;
	
			IF fbXmlSrvReadByAdd.bExecute AND NOT fbXmlSrvReadByAdd.bBusy AND NOT fbXmlSrvReadByAdd.bError 
			AND fbXmlSrvReadByAdd.sFilePath 	= sFilePath_Int
			AND fbXmlSrvReadByAdd.sXPath		= sXPath_Int	THEN
				iCase := 23; // Read Done -> Proceed to clear FB to prepare for Next Cycle (Array)			
				
			ELSIF fbXmlSrvReadByAdd.bError THEN
				udRead_ErrId := fbXmlSrvReadByAdd.nErrId;
				iCase := 99;	// READ ERROR
				iErrorArrayId	:= iArrayId;
			END_IF

	23: 	//  Read - prepare for Next Cycle (Array) 
			
			bReadSt_Int := FALSE;
	
			IF NOT fbXmlSrvReadByAdd.bExecute AND NOT fbXmlSrvReadByAdd.bBusy  THEN
				iCase := 1; // Proceed to Next Cycle (Array)
			END_IF
		
		
	29: // Read - All Done 
		
			bRead_Busy 	:= FALSE;
			bRead_Done 	:= TRUE;
		
	
	99: // Error
	
			bWriteSt_Int 	:= FALSE;
			bReadSt_Int 	:= FALSE;

END_CASE

END_FUNCTION_BLOCK

// ---- FBs/B_JKS_OldFB/Compare/EQ_LT.TcPOU
FUNCTION_BLOCK EQ_LT
VAR_INPUT
	INT_SOURCE_A:INT;
	INT_SOURCE_B:INT;
END_VAR
VAR_OUTPUT
	SIGNAL_BOOL:BOOL;
END_VAR
VAR
	M0: BOOL;
	M1: BOOL;
END_VAR

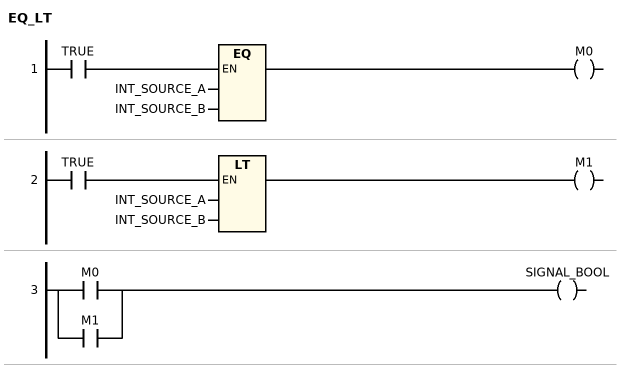
// NETWORK 1
M0 := INT_SOURCE_A = INT_SOURCE_B;

// NETWORK 2
M1 := INT_SOURCE_A < INT_SOURCE_B;

// NETWORK 3
SIGNAL_BOOL := M0 OR M1;

END_FUNCTION_BLOCK

// ---- FBs/B_JKS_OldFB/Compare/LT_GT.TcPOU
FUNCTION_BLOCK LT_GT
VAR_INPUT
	INT_SOURCE_A: INT;
	INT_SOURCE_B: INT;
END_VAR
VAR_OUTPUT
	SIGNAL_BOOL: BOOL;
END_VAR
VAR
	M0: BOOL;
	M1: BOOL;
END_VAR

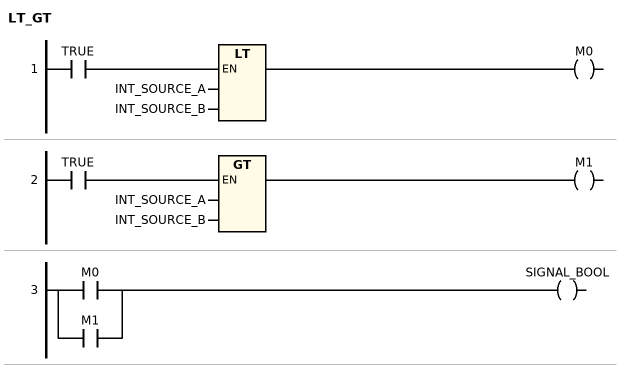
// NETWORK 1
M0 := INT_SOURCE_A < INT_SOURCE_B;

// NETWORK 2
M1 := INT_SOURCE_A > INT_SOURCE_B;

// NETWORK 3
SIGNAL_BOOL := M0 OR M1;

END_FUNCTION_BLOCK

// ---- FBs/B_JKS_OldFB/Compare/SERVO_POS_CONFIRM.TcPOU
FUNCTION_BLOCK SERVO_POS_CONFIRM
VAR_INPUT
	BOOL_JOG_ACTIVE : BOOL;
	UINT_TARGET1 : UINT;
	UINT_TARGET2 : UINT;
	UINT_TARGET3 : UINT;
	UINT_TARGET4 : UINT;
	COUNTER_VALUE : UINT;
	HOMING_READY : BOOL;
END_VAR

VAR_OUTPUT
	TARGET1_CONFIRM_BOOL : BOOL;
	TARGET2_CONFIRM_BOOL : BOOL;
	TARGET3_CONFIRM_BOOL : BOOL;
	TARGET4_CONFIRM_BOOL : BOOL;
END_VAR
VAR
	T1C: BOOL;
	T2C: BOOL;
	T3C: BOOL;
	T4C: BOOL;
END_VAR

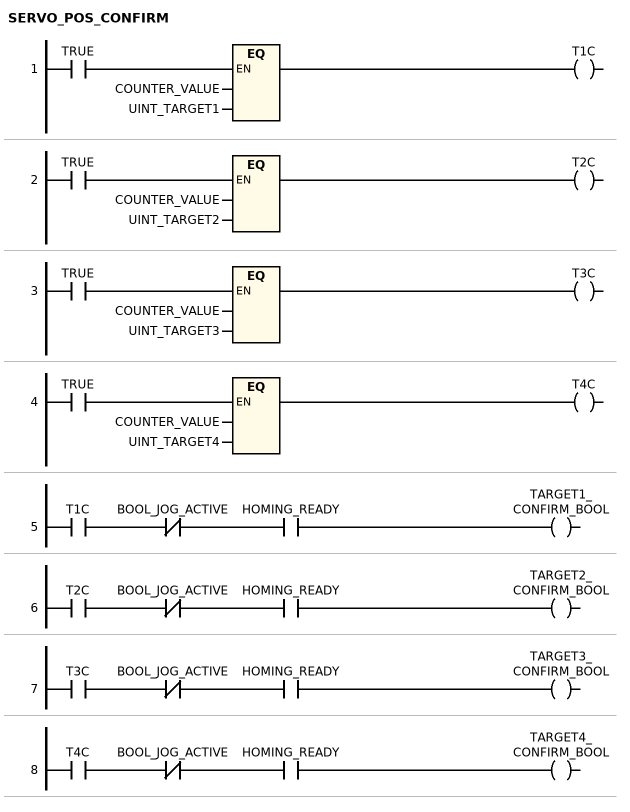
// NETWORK 1
T1C := COUNTER_VALUE = UINT_TARGET1;

// NETWORK 2
T2C := COUNTER_VALUE = UINT_TARGET2;

// NETWORK 3
T3C := COUNTER_VALUE = UINT_TARGET3;

// NETWORK 4
T4C := COUNTER_VALUE = UINT_TARGET4;

// NETWORK 5
TARGET1_CONFIRM_BOOL := T1C AND NOT BOOL_JOG_ACTIVE AND HOMING_READY;

// NETWORK 6
TARGET2_CONFIRM_BOOL := T2C AND NOT BOOL_JOG_ACTIVE AND HOMING_READY;

// NETWORK 7
TARGET3_CONFIRM_BOOL := T3C AND NOT BOOL_JOG_ACTIVE AND HOMING_READY;

// NETWORK 8
TARGET4_CONFIRM_BOOL := T4C AND NOT BOOL_JOG_ACTIVE AND HOMING_READY;

END_FUNCTION_BLOCK

// ---- FBs/B_JKS_OldFB/Controller/GUYSON_PRG_SEL.TcPOU
FUNCTION_BLOCK GUYSON_PRG_SEL
VAR_INPUT

	US_ON_BOOL		:BOOL; 		(*ULTRASONIC ON/OFF BIT*)
	PRG_ADD_INT		:INT;		(*PROGRAM ADDRESS*)


END_VAR
VAR_OUTPUT

	BOOL_US_BIT1		:BOOL; 		(*ULTRASONIC EXT1*)
	BOOL_US_BIT2		:BOOL; 		(*ULTRASONIC EXT2*)
	BOOL_US_BIT3		:BOOL; 		(*ULTRASONIC EXT3*)


END_VAR
VAR
END_VAR

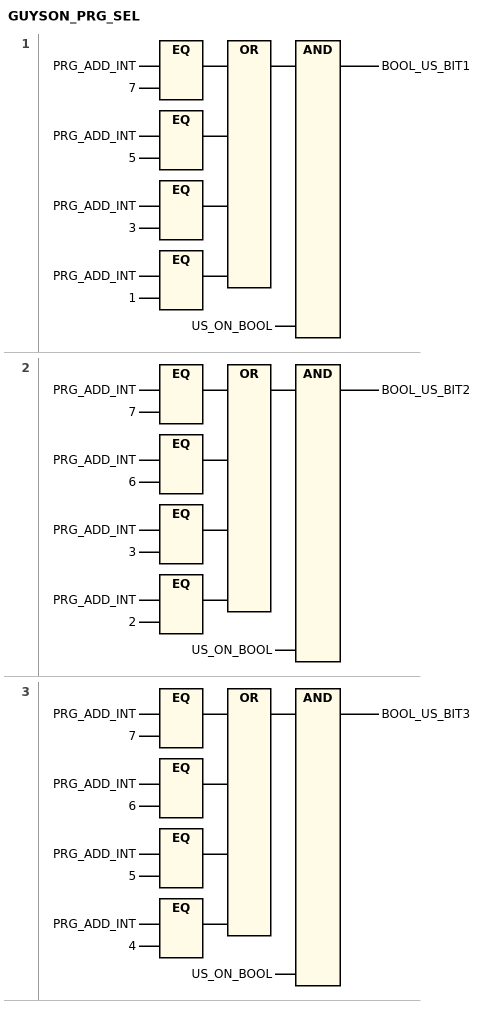
// NETWORK 1
BOOL_US_BIT1 := (PRG_ADD_INT = 7 OR PRG_ADD_INT = 5 OR PRG_ADD_INT = 3 OR PRG_ADD_INT = 1) AND US_ON_BOOL;

// NETWORK 2
BOOL_US_BIT2 := (PRG_ADD_INT = 7 OR PRG_ADD_INT = 6 OR PRG_ADD_INT = 3 OR PRG_ADD_INT = 2) AND US_ON_BOOL;

// NETWORK 3
BOOL_US_BIT3 := (PRG_ADD_INT = 7 OR PRG_ADD_INT = 6 OR PRG_ADD_INT = 5 OR PRG_ADD_INT = 4) AND US_ON_BOOL;

END_FUNCTION_BLOCK

// ---- FBs/B_JKS_OldFB/Controller/MOTION_ACC_DCC.TcPOU
FUNCTION_BLOCK MOTION_ACC_DCC
VAR_INPUT
	BOOL_UP_MOVE : BOOL;
	BOOL_DOWN_MOVE : BOOL;
	UINT_JOG_ACCDCC : UINT;
	UINT_HOME_ACCDCC : UINT;
	UINT_UD_ACCDCC : UINT;
	UINT_AG_ACCDCC : UINT;
	TIME_UD_DLY_ON : TIME;
	BOOL_MANUAL_PG : BOOL;
	BOOL_ORIGIN_COMP : BOOL;
	BOOL_ARM_HOME_READY : BOOL;
	STRING_CURRENT_PG : STRING;
	STRING_MAN_JOG_V_PG : STRING;
	STRING_MAN_POS_V_PG : STRING;
	STRING_MAN_JOG_H_PG : STRING;
	STRING_MAN_POS_H_PG : STRING;
END_VAR
VAR_OUTPUT

	UP_MOVE_ST_BOOL : BOOL;
	DOWN_MOVE_ST_BOOL : BOOL;
	ACC_UINT : UINT;
	DCC_UINT : UINT;

END_VAR
VAR
	T1: TON;
	T1COUNT: TIME;
	T2: TON;
	T2COUNT: TIME;
	MANJOGH: BOOL;
	MANJOGV: BOOL;
	MANPOSH: BOOL;
	MANPOSV: BOOL;
END_VAR
VAR // added by the converter: edge detectors and wires of the graphical bodies
    _w1, _w4, _w7, _w10 : BOOL;
    _w2, _w3, _w5, _w6, _w8, _w9, _w11, _w12 : UINT;
END_VAR

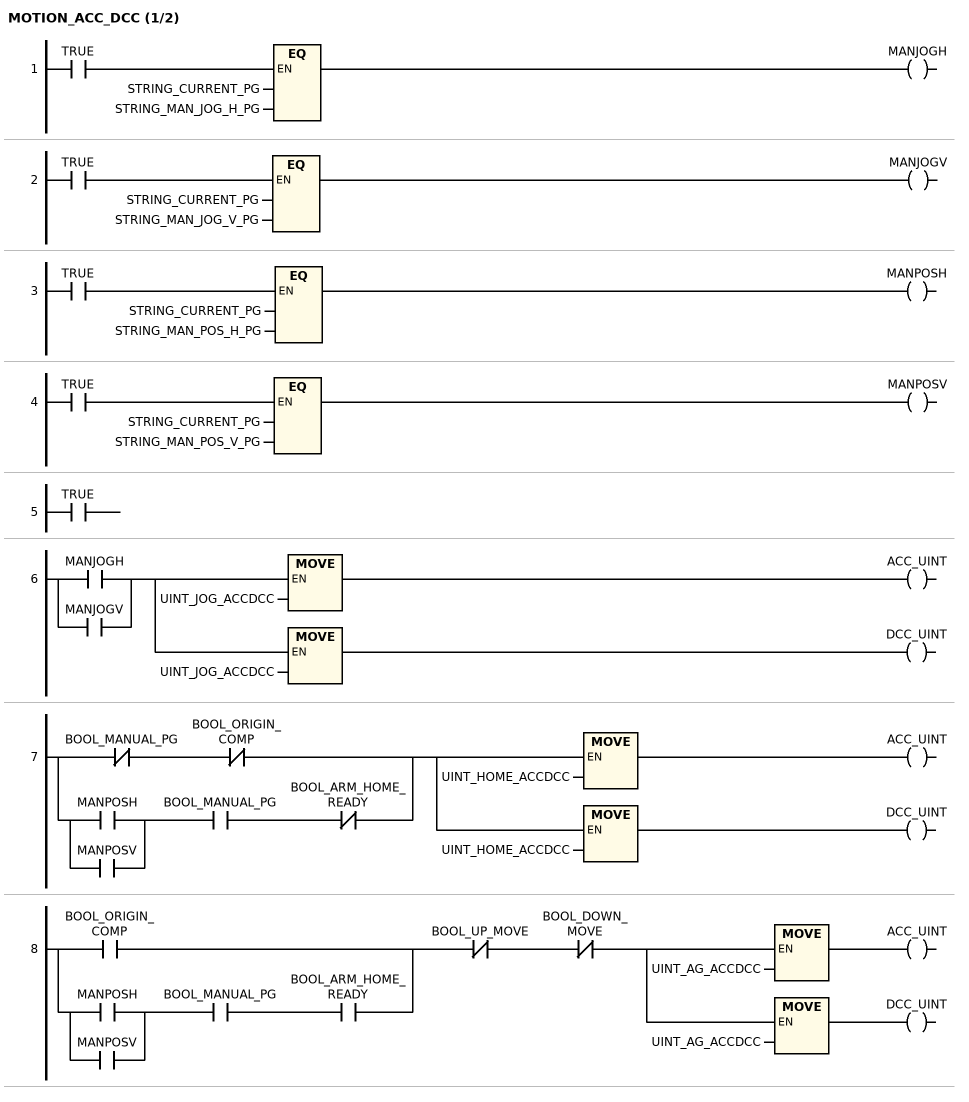
// NETWORK 1
MANJOGH := STRING_CURRENT_PG = STRING_MAN_JOG_H_PG;

// NETWORK 2
MANJOGV := STRING_CURRENT_PG = STRING_MAN_JOG_V_PG;

// NETWORK 3
MANPOSH := STRING_CURRENT_PG = STRING_MAN_POS_H_PG;

// NETWORK 4
MANPOSV := STRING_CURRENT_PG = STRING_MAN_POS_V_PG;

// NETWORK 5

// NETWORK 6
_w1 := MANJOGH OR MANJOGV;
IF _w1 THEN _w2 := UINT_JOG_ACCDCC; END_IF
ACC_UINT := _w2;
IF _w1 THEN _w3 := UINT_JOG_ACCDCC; END_IF
DCC_UINT := _w3;

// NETWORK 7
_w4 := NOT BOOL_MANUAL_PG AND NOT BOOL_ORIGIN_COMP OR (MANPOSH OR MANPOSV) AND BOOL_MANUAL_PG AND NOT BOOL_ARM_HOME_READY;
IF _w4 THEN _w5 := UINT_HOME_ACCDCC; END_IF
ACC_UINT := _w5;
IF _w4 THEN _w6 := UINT_HOME_ACCDCC; END_IF
DCC_UINT := _w6;

// NETWORK 8
_w7 := (BOOL_ORIGIN_COMP OR (MANPOSH OR MANPOSV) AND BOOL_MANUAL_PG AND BOOL_ARM_HOME_READY) AND NOT BOOL_UP_MOVE AND NOT BOOL_DOWN_MOVE;
IF _w7 THEN _w8 := UINT_AG_ACCDCC; END_IF
ACC_UINT := _w8;
IF _w7 THEN _w9 := UINT_AG_ACCDCC; END_IF
DCC_UINT := _w9;

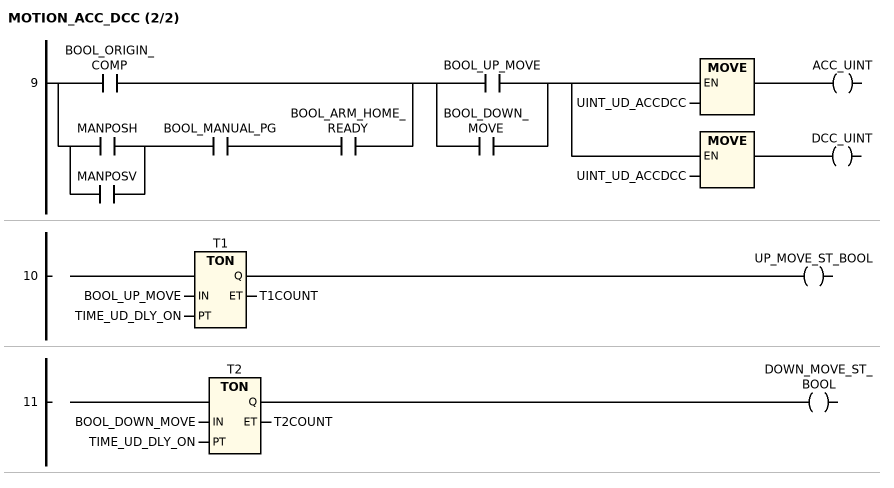
// NETWORK 9
_w10 := (BOOL_ORIGIN_COMP OR (MANPOSH OR MANPOSV) AND BOOL_MANUAL_PG AND BOOL_ARM_HOME_READY) AND (BOOL_UP_MOVE OR BOOL_DOWN_MOVE);
IF _w10 THEN _w11 := UINT_UD_ACCDCC; END_IF
ACC_UINT := _w11;
IF _w10 THEN _w12 := UINT_UD_ACCDCC; END_IF
DCC_UINT := _w12;

// NETWORK 10
T1(IN := BOOL_UP_MOVE, PT := TIME_UD_DLY_ON, ET => T1COUNT); // TON
UP_MOVE_ST_BOOL := T1.Q;

// NETWORK 11
T2(IN := BOOL_DOWN_MOVE, PT := TIME_UD_DLY_ON, ET => T2COUNT); // TON
DOWN_MOVE_ST_BOOL := T2.Q;

END_FUNCTION_BLOCK

// ---- FBs/B_JKS_OldFB/Controller/TEMP_CTRL_ON_OFF.TcPOU
FUNCTION_BLOCK TEMP_CTRL_ON_OFF
VAR_INPUT
	REAL_SV			: REAL;
	REAL_HYS			: REAL;
	REAL_HAL			: REAL;
	REAL_T_READY		: REAL; (*Value set base on -X*)
	TOutOfRangeNegative	: REAL; (*Value set base on +/- X*)
	TOutOfRangePositive	: REAL;
END_VAR


VAR_OUTPUT
	REAL_PV : REAL;
	OUT_BOOL: BOOL;
	HAL_BOOL: BOOL;
	T_READY_BOOL: BOOL;
	T_OutOfRange_BOOL : BOOL;
END_VAR

VAR
	TEMP_PV	AT %I*	: INT;
	TREADY_TEMP: REAL;
	HYS_TEMP: REAL;
	ALWAYS_OFF: BOOL;
	ALWAYS_ON_BOOL: BOOL;
	T1: TON;
	PLS1: R_TRIG;
	RS1: RS;

END_VAR

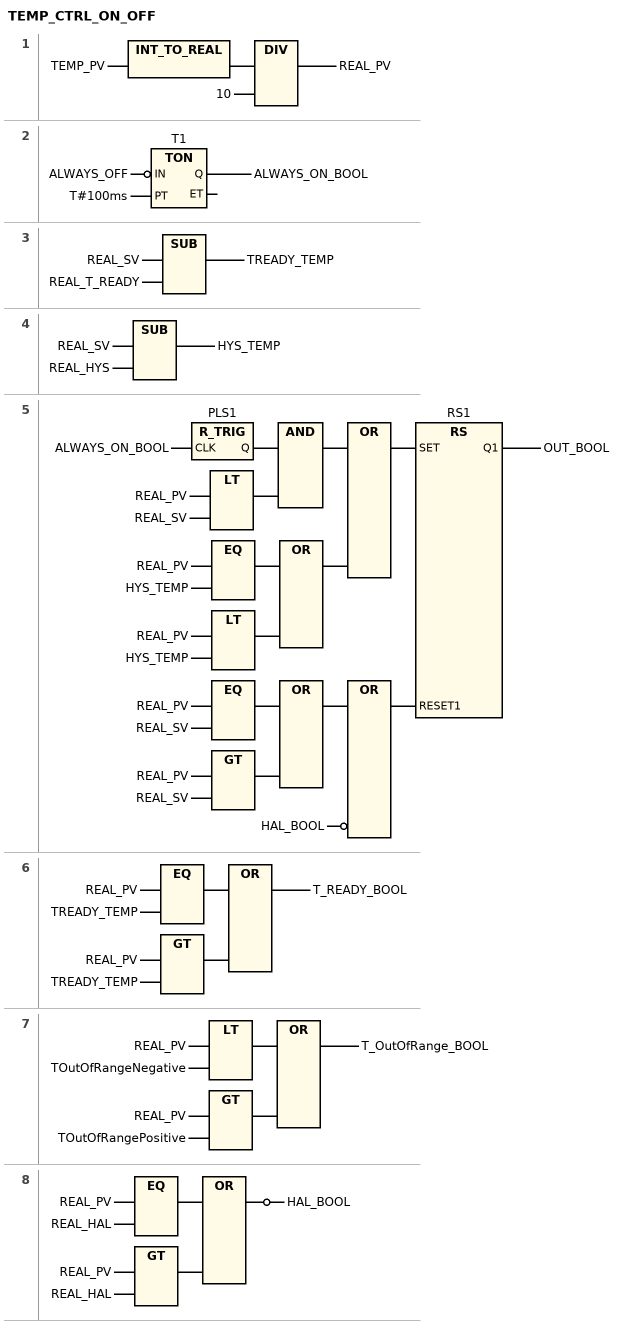
// NETWORK 1
REAL_PV := INT_TO_REAL(TEMP_PV) / 10;

// NETWORK 2
T1(IN := NOT ALWAYS_OFF, PT := T#100ms); // TON
ALWAYS_ON_BOOL := T1.Q;

// NETWORK 3
TREADY_TEMP := REAL_SV - REAL_T_READY;

// NETWORK 4
HYS_TEMP := REAL_SV - REAL_HYS;

// NETWORK 5
PLS1(CLK := ALWAYS_ON_BOOL); // R_TRIG
RS1(SET := PLS1.Q AND REAL_PV < REAL_SV OR (REAL_PV = HYS_TEMP OR REAL_PV < HYS_TEMP), RESET1 := (REAL_PV = REAL_SV OR REAL_PV > REAL_SV) OR NOT HAL_BOOL); // RS
OUT_BOOL := RS1.Q1;

// NETWORK 6
T_READY_BOOL := REAL_PV = TREADY_TEMP OR REAL_PV > TREADY_TEMP;

// NETWORK 7
T_OutOfRange_BOOL := REAL_PV < TOutOfRangeNegative OR REAL_PV > TOutOfRangePositive;

// NETWORK 8
HAL_BOOL := NOT (REAL_PV = REAL_HAL OR REAL_PV > REAL_HAL);

END_FUNCTION_BLOCK

// ---- FBs/B_JKS_OldFB/Controller/TEMP_CTRL_ON_OFF_EXT.TcPOU
FUNCTION_BLOCK TEMP_CTRL_ON_OFF_EXT
VAR_INPUT
	REAL_SV			: REAL;
	REAL_HYS			: REAL;
	REAL_HAL			: REAL;
	REAL_T_READY		: REAL; (*Value set base on -X*)
	TOutOfRangeNegative	: REAL; (*Value set base on +/- X*)
	TOutOfRangePositive	: REAL;
	INT_PV				: INT;

END_VAR


VAR_OUTPUT
	REAL_PV : REAL;
	OUT_BOOL: BOOL;
	HAL_BOOL: BOOL;
	T_READY_BOOL: BOOL;
	T_OutOfRange_BOOL : BOOL;
END_VAR

VAR

	TREADY_TEMP: REAL;
	HYS_TEMP: REAL;
	ALWAYS_OFF: BOOL;
	ALWAYS_ON_BOOL: BOOL;
	T1: TON;
	PLS1: R_TRIG;
	RS1: RS;

END_VAR

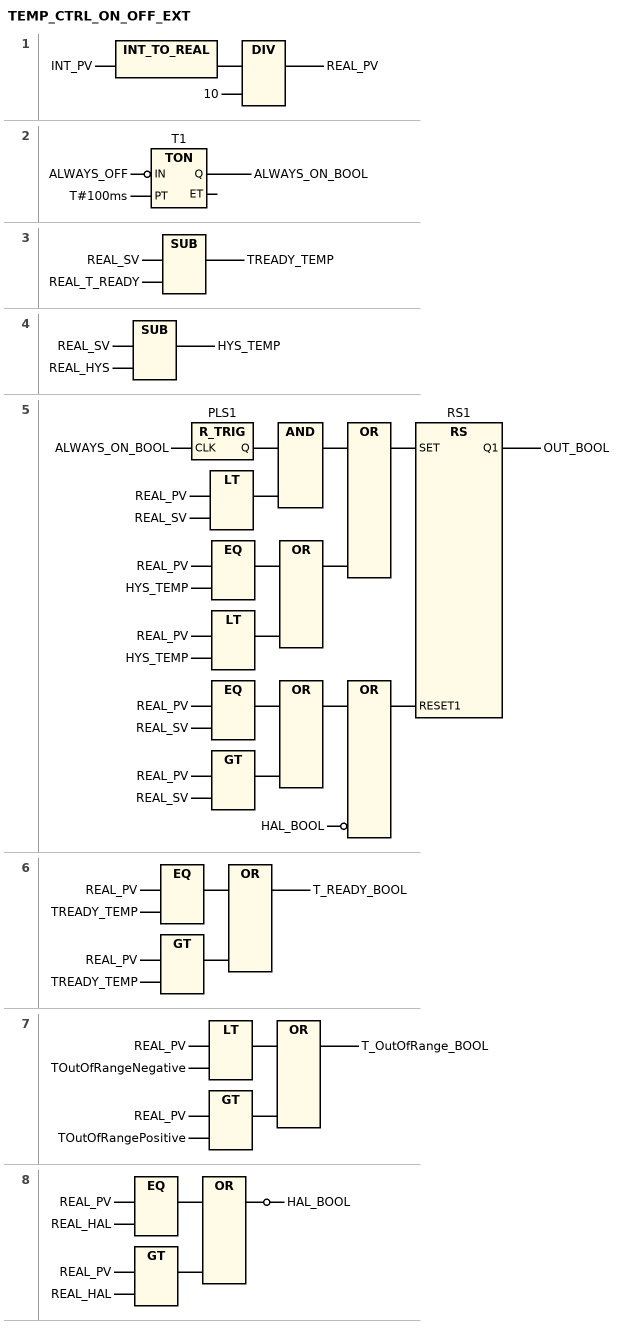
// NETWORK 1
REAL_PV := INT_TO_REAL(INT_PV) / 10;

// NETWORK 2
T1(IN := NOT ALWAYS_OFF, PT := T#100ms); // TON
ALWAYS_ON_BOOL := T1.Q;

// NETWORK 3
TREADY_TEMP := REAL_SV - REAL_T_READY;

// NETWORK 4
HYS_TEMP := REAL_SV - REAL_HYS;

// NETWORK 5
PLS1(CLK := ALWAYS_ON_BOOL); // R_TRIG
RS1(SET := PLS1.Q AND REAL_PV < REAL_SV OR (REAL_PV = HYS_TEMP OR REAL_PV < HYS_TEMP), RESET1 := (REAL_PV = REAL_SV OR REAL_PV > REAL_SV) OR NOT HAL_BOOL); // RS
OUT_BOOL := RS1.Q1;

// NETWORK 6
T_READY_BOOL := REAL_PV = TREADY_TEMP OR REAL_PV > TREADY_TEMP;

// NETWORK 7
T_OutOfRange_BOOL := REAL_PV < TOutOfRangeNegative OR REAL_PV > TOutOfRangePositive;

// NETWORK 8
HAL_BOOL := NOT (REAL_PV = REAL_HAL OR REAL_PV > REAL_HAL);

END_FUNCTION_BLOCK

// ---- FBs/B_JKS_OldFB/Converter/DC_PID_FB.TcPOU
FUNCTION_BLOCK DC_PID_FB
VAR_INPUT
	BOOL_LOW_FLOW_EN : BOOL;
	INT_HIGH_FLOW_LPM : INT;
	INT_LOW_FLOW_LPM : INT;
	INT_H_L_FLOW_RATIO : INT;
	INT_D1_LPM : INT;
	INT_D2_LPM : INT;
	INT_D3_LPM : INT;
	INT_D4_RAW : INT;
	INT_D5_RAW : INT;
	INT_D6_RAW : INT;
	INT_D1_RATIO : INT;
	INT_D2_RATIO : INT;
	INT_D3_RATIO : INT;
	INT_D4_RATIO : INT;
	INT_D5_RATIO : INT;
	INT_D6_RATIO : INT;

END_VAR

VAR_OUTPUT

	PID_FLOW_RAW : INT;
	D1_RAW_INT : INT;
	D2_RAW_INT : INT;
	D3_RAW_INT : INT;
	D4_LPM_INT : INT;
	D5_LPM_INT : INT;
	D6_LPM_INT : INT;

END_VAR
VAR
	D5EN: BOOL;
	D4EN: BOOL;
	D6EN: BOOL;
	D4REN: BOOL;
	D5REN: BOOL;
	D6REN: BOOL;
END_VAR

(*

Thats 2 program in one function block

1st Program:- 
- Let user able to select High/low flow by trigger bit "BOOL_LOW_FLOW_EN"

	Sequence detail: 
	-If "BOOL_LOW_FLOW_EN" OFF, "INT_HIGH_FLOW_LPM" will MULTIPLY "INT_H_L_FLOW_RATIO" then Feed into "PID_FLOW_RAW".
	-If "BOOL_LOW_FLOW_EN" ON, "INT_LOW_FLOW_LPM" will MULTIPLY "INT_H_L_FLOW_RATIO" then Feed into "PID_FLOW_RAW".
	-"PID_FLOW_RAW should connect direct to ANALOG OUTPUT CARD CHANNEL.


2nd Program:-
-Become Converter. Able to convert 3 types of LPM reading to RAW reading by MULTIPLY the preset RATIO.
-Become Converter. Able to convert 3 types of RAW reading to LPM reading by DIVIDE the preset RATIO.

	Sequence detail:
	-Once detected INT_D1_LPM have value (Not "0") and INT_D1_RATIO have value (Not "0") -> Program will enable and MULTIPLY "INT_D1_LPM" with "INT_D1_RATIO" and feed to "D1_RAW_INT"
	-INT_D2_LPM, INT_D2_RATIO and D2_RAW_INT function same as above (D1)
	-INT_D3_LPM, INT_D3_RATIO and D3_RAW_INT function same as above (D1)
	-Once detected INT_D4_RAW have value (Not "0") and INT_D4_RATIO have value (Not "0") -> Program will enable and DIVIDE "INT_D4_RAW" with "INT_D4_RATIO" and feed to "D4_LPM_INT"
	-INT_D5_RAW, INT_D5_RATIO and D5_LPM_INT function same as above (D4)
	-INT_D6_RAW, INT_D6_RATIO and D6_LPM_INT function same as above (D4)

*)
VAR // added by the converter: edge detectors and wires of the graphical bodies
    _w1, _w2, _w3, _w4, _w5 : INT;
END_VAR

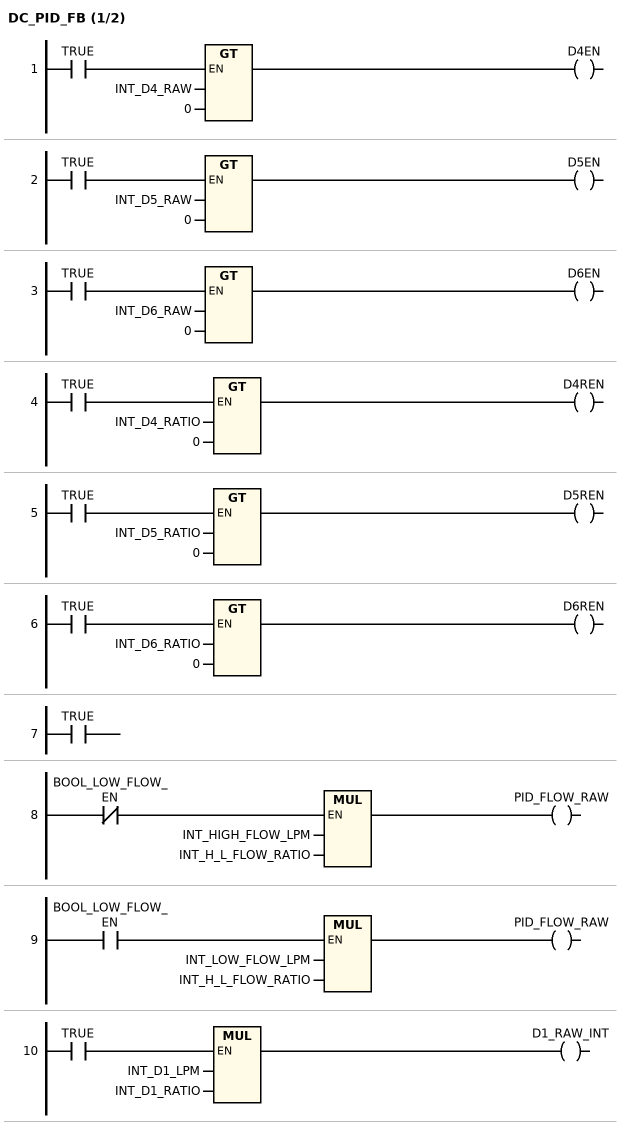
// NETWORK 1
D4EN := INT_D4_RAW > 0;

// NETWORK 2
D5EN := INT_D5_RAW > 0;

// NETWORK 3
D6EN := INT_D6_RAW > 0;

// NETWORK 4
D4REN := INT_D4_RATIO > 0;

// NETWORK 5
D5REN := INT_D5_RATIO > 0;

// NETWORK 6
D6REN := INT_D6_RATIO > 0;

// NETWORK 7

// NETWORK 8
IF NOT BOOL_LOW_FLOW_EN THEN _w1 := INT_HIGH_FLOW_LPM * INT_H_L_FLOW_RATIO; END_IF
PID_FLOW_RAW := _w1;

// NETWORK 9
IF BOOL_LOW_FLOW_EN THEN _w2 := INT_LOW_FLOW_LPM * INT_H_L_FLOW_RATIO; END_IF
PID_FLOW_RAW := _w2;

// NETWORK 10
D1_RAW_INT := INT_D1_LPM * INT_D1_RATIO;

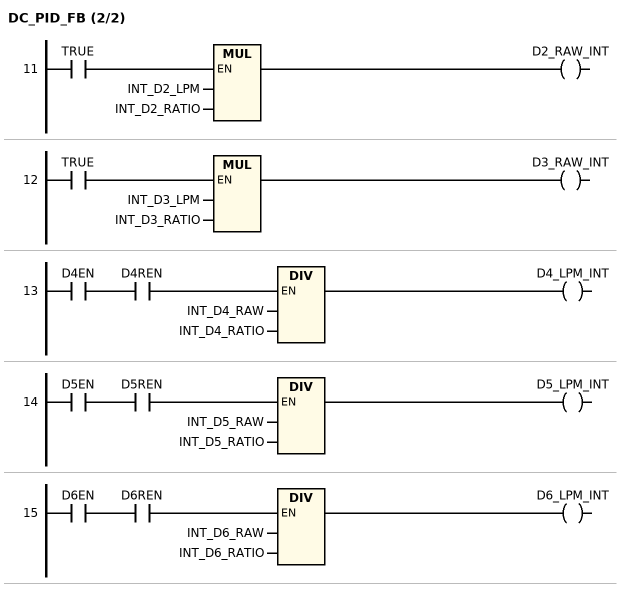
// NETWORK 11
D2_RAW_INT := INT_D2_LPM * INT_D2_RATIO;

// NETWORK 12
D3_RAW_INT := INT_D3_LPM * INT_D3_RATIO;

// NETWORK 13
IF D4EN AND D4REN THEN _w3 := INT_D4_RAW / INT_D4_RATIO; END_IF
D4_LPM_INT := _w3;

// NETWORK 14
IF D5EN AND D5REN THEN _w4 := INT_D5_RAW / INT_D5_RATIO; END_IF
D5_LPM_INT := _w4;

// NETWORK 15
IF D6EN AND D6REN THEN _w5 := INT_D6_RAW / INT_D6_RATIO; END_IF
D6_LPM_INT := _w5;

END_FUNCTION_BLOCK

// ---- FBs/B_JKS_OldFB/Converter/JOG_CONV.TcPOU
FUNCTION_BLOCK JOG_CONV
VAR_INPUT
	BOOL_FWD_JOG : BOOL;
	BOOL_RWD_JOG : BOOL;
	UINT_JOG_SPD_MM : UINT;
	TIME_JOG_DELAY : TIME;
	UINT_PLS_RATIO : UINT;

END_VAR
VAR_OUTPUT
	JOG_ACTIVE_BOOL : BOOL;
	JOG_SPD_UINT : UINT;


END_VAR
VAR
	VUINT: UINT;
	T1: TON;
	TI: TIME;
	JSPD_PLS: UINT;
END_VAR
VAR // added by the converter: edge detectors and wires of the graphical bodies
    _w1, _w2 : UINT;
END_VAR

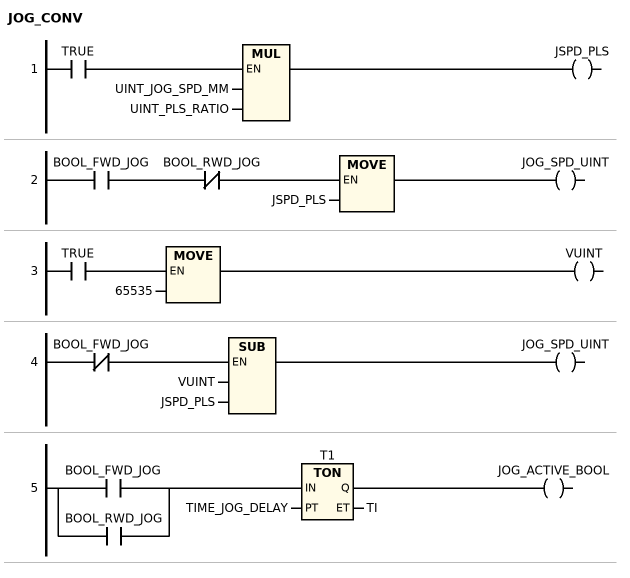
// NETWORK 1
JSPD_PLS := UINT_JOG_SPD_MM * UINT_PLS_RATIO;

// NETWORK 2
IF BOOL_FWD_JOG AND NOT BOOL_RWD_JOG THEN _w1 := JSPD_PLS; END_IF
JOG_SPD_UINT := _w1;

// NETWORK 3
VUINT := 65535;

// NETWORK 4
IF NOT BOOL_FWD_JOG THEN _w2 := VUINT - JSPD_PLS; END_IF
JOG_SPD_UINT := _w2;

// NETWORK 5
T1(IN := BOOL_FWD_JOG OR BOOL_RWD_JOG, PT := TIME_JOG_DELAY, ET => TI); // TON
JOG_ACTIVE_BOOL := T1.Q;

END_FUNCTION_BLOCK

// ---- FBs/B_JKS_OldFB/Converter/MM_TO_PLS.TcPOU
FUNCTION_BLOCK MM_TO_PLS
VAR_INPUT
	UINT_PLS_RATIO : UINT;
	UINT_TARGET1_MM : UINT;
	UINT_VEL1_MM : UINT;
	UINT_TARGET2_MM : UINT;
	UINT_VEL2_MM : UINT;
	UINT_TARGET3_MM : UINT;
	UINT_VEL3_MM : UINT;
	UINT_TARGET4_MM : UINT;
	UINT_VEL4_MM : UINT;
	UINT_JOG_2SPD_MM : UINT;
END_VAR

VAR_OUTPUT
	TARGET1_WR_UINT : UINT;
	VEL1_WR_UINT : UINT;
	TARGET2_WR_UINT : UINT;
	VEL2_WR_UINT : UINT;
	TARGET3_WR_UINT : UINT;
	VEL3_WR_UINT : UINT;
	TARGET4_WR_UINT : UINT;
	VEL4_WR_UINT : UINT;
	JOG_2SPD_UINT : UINT;

END_VAR

VAR
END_VAR

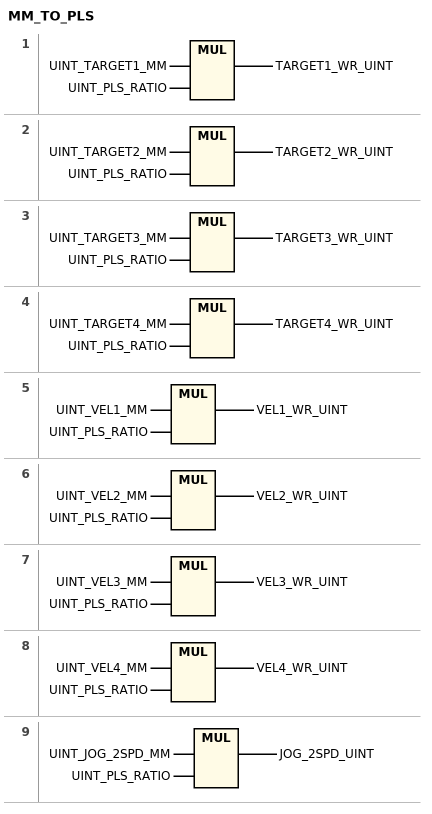
// NETWORK 1
TARGET1_WR_UINT := UINT_TARGET1_MM * UINT_PLS_RATIO;

// NETWORK 2
TARGET2_WR_UINT := UINT_TARGET2_MM * UINT_PLS_RATIO;

// NETWORK 3
TARGET3_WR_UINT := UINT_TARGET3_MM * UINT_PLS_RATIO;

// NETWORK 4
TARGET4_WR_UINT := UINT_TARGET4_MM * UINT_PLS_RATIO;

// NETWORK 5
VEL1_WR_UINT := UINT_VEL1_MM * UINT_PLS_RATIO;

// NETWORK 6
VEL2_WR_UINT := UINT_VEL2_MM * UINT_PLS_RATIO;

// NETWORK 7
VEL3_WR_UINT := UINT_VEL3_MM * UINT_PLS_RATIO;

// NETWORK 8
VEL4_WR_UINT := UINT_VEL4_MM * UINT_PLS_RATIO;

// NETWORK 9
JOG_2SPD_UINT := UINT_JOG_2SPD_MM * UINT_PLS_RATIO;

END_FUNCTION_BLOCK

// ---- FBs/B_JKS_OldFB/Guyson/GUYSON_AI_CTRL.TcPOU
FUNCTION_BLOCK GUYSON_AI_CTRL
VAR_INPUT

	BOOL_ST :BOOL; (*Analog Data Collection Start Bit*)
	INT_M1_AI :INT; (*Guyson Generator Master 1 Analog Input Data*)
	INT_M2_AI :INT; (*Guyson Generator Master 2 Analog Input Data*)
	TIME_REFRESH :TIME; (*Refresh Time assigned*)
	TIME_DATA_COLLECT :TIME; (*Delay time for data collection for stability improvement, This data must be ALWAYS "Half" or below from "TIME_REFRESH" SetPoint *)

END_VAR

VAR_OUTPUT

	M1CH1_INT :INT; (*ANALOG READING OF MASTER1-CHANNEL1*)
	M1CH2_INT :INT; (*ANALOG READING OF MASTER1-CHANNEL2*)
	S1CH1_INT :INT; (*ANALOG READING OF SLAVE1-CHANNEL1*)
	M2CH1_INT :INT; (*ANALOG READING OF MASTER2-CHANNEL1*)
	M2CH2_INT :INT; (*ANALOG READING OF MASTER2-CHANNEL2*)
	S2CH1_INT :INT; (*ANALOG READING OF SLAVE2-CHANNEL1*)
	M1_PIN1_DO_BOOL :BOOL; (*GUYSON MASTER 1 SCADA CONNECTOR PIN 1 (A0) CONNECTION OUTPUT FOR MODULE SELECTION*)
	M1_PIN7_DO_BOOL :BOOL; (*GUYSON MASTER 1 SCADA CONNECTOR PIN 7 (A3) CONNECTION OUTPUT FOR IDENTITY SELECTION*)
	M2_PIN1_DO_BOOL :BOOL; (*GUYSON MASTER 2 SCADA CONNECTOR PIN 1 (A0) CONNECTION OUTPUT FOR MODULE SELECTION*)
	M2_PIN7_DO_BOOL :BOOL; (*GUYSON MASTER 2 SCADA CONNECTOR PIN 7 (A3) CONNECTION OUTPUT FOR IDENTITY SELECTION*)
	IT1AOUT_BOOL: BOOL;
	IT2AOUT_BOOL: BOOL;
	IT3AOUT_BOOL: BOOL;
	IT1BOUT_BOOL: BOOL;
	IT2BOUT_BOOL: BOOL;
	IT3BOUT_BOOL: BOOL;





END_VAR
VAR
	IT1A: TON;
	IT2A: TON;
	IT3A: TON;
	IT1B: TON;
	IT2B: TON;
	IT3B: TON;


	M1CH1BOOLOUT: BOOL;
	M1CH2BOOLOUT: BOOL;
	S1CH1BOOLOUT: BOOL;
	M2CH1BOOLOUT: BOOL;
	M2CH2BOOLOUT: BOOL;
	S2CH1BOOLOUT: BOOL;

END_VAR
VAR // added by the converter: edge detectors and wires of the graphical bodies
    _w1, _w2, _w3 : BOOL;
    _w4, _w5, _w6, _w7, _w8, _w9 : INT;
END_VAR

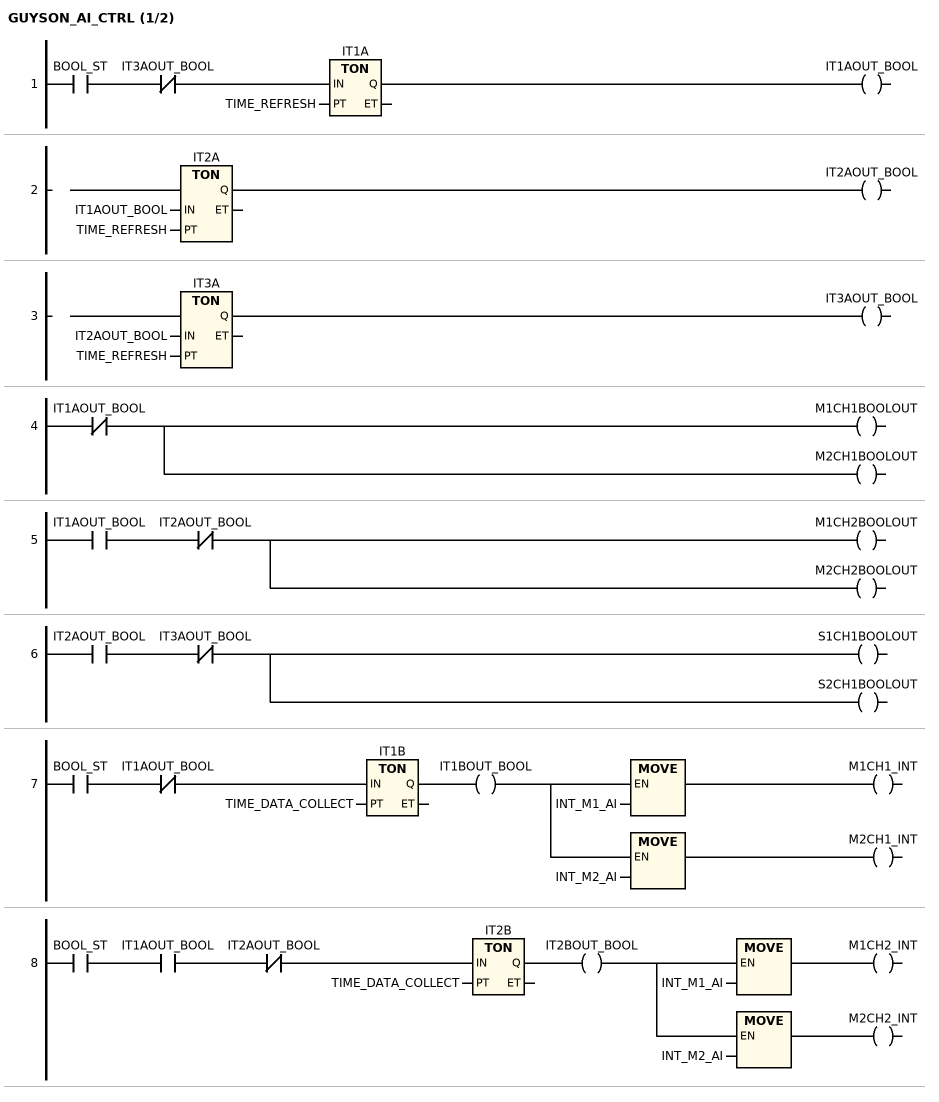
// NETWORK 1
IT1A(IN := BOOL_ST AND NOT IT3AOUT_BOOL, PT := TIME_REFRESH); // TON
IT1AOUT_BOOL := IT1A.Q;

// NETWORK 2
IT2A(IN := IT1AOUT_BOOL, PT := TIME_REFRESH); // TON
IT2AOUT_BOOL := IT2A.Q;

// NETWORK 3
IT3A(IN := IT2AOUT_BOOL, PT := TIME_REFRESH); // TON
IT3AOUT_BOOL := IT3A.Q;

// NETWORK 4
_w1 := NOT IT1AOUT_BOOL;
M1CH1BOOLOUT := _w1;
M2CH1BOOLOUT := _w1;

// NETWORK 5
_w2 := IT1AOUT_BOOL AND NOT IT2AOUT_BOOL;
M1CH2BOOLOUT := _w2;
M2CH2BOOLOUT := _w2;

// NETWORK 6
_w3 := IT2AOUT_BOOL AND NOT IT3AOUT_BOOL;
S1CH1BOOLOUT := _w3;
S2CH1BOOLOUT := _w3;

// NETWORK 7
IT1B(IN := BOOL_ST AND NOT IT1AOUT_BOOL, PT := TIME_DATA_COLLECT); // TON
IT1BOUT_BOOL := IT1B.Q;
IF IT1B.Q THEN _w4 := INT_M1_AI; END_IF
M1CH1_INT := _w4;
IF IT1B.Q THEN _w5 := INT_M2_AI; END_IF
M2CH1_INT := _w5;

// NETWORK 8
IT2B(IN := BOOL_ST AND IT1AOUT_BOOL AND NOT IT2AOUT_BOOL, PT := TIME_DATA_COLLECT); // TON
IT2BOUT_BOOL := IT2B.Q;
IF IT2B.Q THEN _w6 := INT_M1_AI; END_IF
M1CH2_INT := _w6;
IF IT2B.Q THEN _w7 := INT_M2_AI; END_IF
M2CH2_INT := _w7;

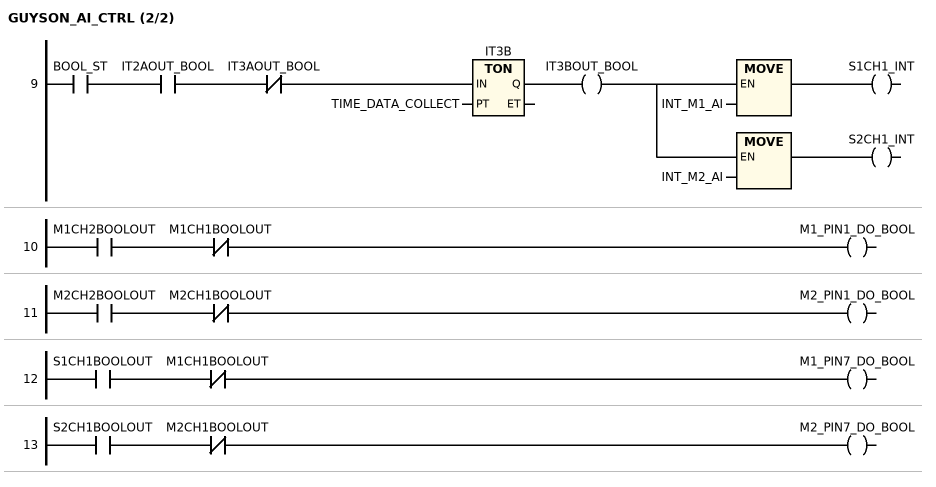
// NETWORK 9
IT3B(IN := BOOL_ST AND IT2AOUT_BOOL AND NOT IT3AOUT_BOOL, PT := TIME_DATA_COLLECT); // TON
IT3BOUT_BOOL := IT3B.Q;
IF IT3B.Q THEN _w8 := INT_M1_AI; END_IF
S1CH1_INT := _w8;
IF IT3B.Q THEN _w9 := INT_M2_AI; END_IF
S2CH1_INT := _w9;

// NETWORK 10
M1_PIN1_DO_BOOL := M1CH2BOOLOUT AND NOT M1CH1BOOLOUT;

// NETWORK 11
M2_PIN1_DO_BOOL := M2CH2BOOLOUT AND NOT M2CH1BOOLOUT;

// NETWORK 12
M1_PIN7_DO_BOOL := S1CH1BOOLOUT AND NOT M1CH1BOOLOUT;

// NETWORK 13
M2_PIN7_DO_BOOL := S2CH1BOOLOUT AND NOT M2CH1BOOLOUT;

END_FUNCTION_BLOCK

// ---- FBs/B_JKS_OldFB/Guyson/GUYSON_AI_RawToWatt.TcPOU
FUNCTION_BLOCK GUYSON_AI_RawToWatt
VAR_INPUT

	iAI1raw : INT;				(* 1st Raw Data From Analog Input*)
	iAI2raw : INT;				(* 2nd Raw Data From Analog Input*)
	iAI3raw : INT;				(* 3rd Raw Data From Analog Input*)
	iAI4raw : INT;				(* 4th Raw Data From Analog Input*)
	iAI5raw : INT;				(* 5th Raw Data From Analog Input*)
	iAI6raw : INT;				(* 6th Raw Data From Analog Input*)
	PercentBase : BOOL;		(* The PV will shown Percentage if this Bit is "ON"*)
	WattBase : BOOL;			(* The PV will shown Wattage if this Bit is "ON"*)
	MaxWatt : INT;			(* Defined Max Watt of Generator, Usually is 700W*)

END_VAR
VAR_OUTPUT

	iAI1Value : INT;			(*PV for 1st Data, either Watt or Percent is depend on Base Setting*)
	iAI2Value : INT;			(*PV for 2nd Data, either Watt or Percent is depend on Base Setting*)
	iAI3Value : INT;			(*PV for 3rd Data, either Watt or Percent is depend on Base Setting*)
	iAI4Value : INT;			(*PV for 4th Data, either Watt or Percent is depend on Base Setting*)
	iAI5Value : INT;			(*PV for 5th Data, either Watt or Percent is depend on Base Setting*)
	iAI6Value : INT;			(*PV for 6th Data, either Watt or Percent is depend on Base Setting*)

END_VAR
VAR
	iAI1f: LREAL;
	iAI2f: LREAL;
	iAI3f: LREAL;
	iAI4f: LREAL;
	iAI5f: LREAL;
	iAI6f: LREAL;

	iAI1_Wf: LREAL;
	iAI2_Wf: LREAL;
	iAI3_Wf: LREAL;
	iAI4_Wf: LREAL;
	iAI5_Wf: LREAL;
	iAI6_Wf: LREAL;

	n : INT;

	WRatio: INT;
END_VAR

iAI1f := INT_TO_LREAL (iAI1raw);
iAI2f := INT_TO_LREAL (iAI2raw);
iAI3f := INT_TO_LREAL (iAI3raw);
iAI4f := INT_TO_LREAL (iAI4raw);
iAI5f := INT_TO_LREAL (iAI5raw);
iAI6f := INT_TO_LREAL (iAI6raw);


(*Program to select Watt Base or Percent Base*)

IF PercentBase AND NOT WattBase THEN
n := 11;
END_IF

IF WattBase AND NOT PercentBase THEN
n := 10;
END_IF

IF NOT PercentBase AND NOT WattBase THEN
n := 0;
END_IF

IF PercentBase AND WattBase THEN
n:= 0;
END_IF

CASE n OF

0:; (*No Calculation*)


10: (*Watt Base Calculation *)

iAI1_Wf	:= (iAI1f / 3276.7) * (iAI1f / 3276.7) *20;
iAI2_Wf	:= (iAI2f / 3276.7) * (iAI2f / 3276.7) *20;
iAI3_Wf	:= (iAI3f / 3276.7) * (iAI3f / 3276.7) *20;
iAI4_Wf	:= (iAI4f / 3276.7) * (iAI4f / 3276.7) *20;
iAI5_Wf	:= (iAI5f / 3276.7) * (iAI5f / 3276.7) *20;
iAI6_Wf	:= (iAI6f / 3276.7) * (iAI6f / 3276.7) *20;


11: (*Percent Base Calculation*)


WRatio := MaxWatt/100;


iAI1_Wf	:= ((iAI1f / 3276.7) * (iAI1f / 3276.7) *20)/WRatio;
iAI2_Wf	:= ((iAI2f / 3276.7) * (iAI2f / 3276.7) *20)/WRatio;
iAI3_Wf	:= ((iAI3f / 3276.7) * (iAI3f / 3276.7) *20)/WRatio;
iAI4_Wf	:= ((iAI4f / 3276.7) * (iAI4f / 3276.7) *20)/WRatio;
iAI5_Wf	:= ((iAI5f / 3276.7) * (iAI5f / 3276.7) *20)/WRatio;
iAI6_Wf	:= ((iAI6f / 3276.7) * (iAI6f / 3276.7) *20)/WRatio;

END_CASE

iAI1Value := LREAL_TO_INT (iAI1_Wf);
iAI2Value := LREAL_TO_INT (iAI2_Wf);
iAI3Value := LREAL_TO_INT (iAI3_Wf);
iAI4Value := LREAL_TO_INT (iAI4_Wf);
iAI5Value := LREAL_TO_INT (iAI5_Wf);
iAI6Value := LREAL_TO_INT (iAI6_Wf);

END_FUNCTION_BLOCK

// ---- FBs/B_JKS_OldFB/Guyson/GUYSON_AI_WattToRaw.TcPOU
FUNCTION_BLOCK GUYSON_AI_WattToRaw
VAR_INPUT

	iAI1SP : INT;			(* 1st SetPoint Data*)
	iAI2SP : INT;			(* 2nd SetPoint Data*)
	iAI3SP : INT;			(* 3rd SetPoint Data*)
	iAI4SP : INT;			(* 4th SetPoint Data*)
	iAI5SP : INT;			(* 5th SetPoint Data*)
	iAI6SP : INT;			(* 6th SetPoint Data*)
	PercentBase : BOOL;	(* The PV will shown Percentage if this Bit is "ON"*)
	WattBase: BOOL;		(* The PV will shown Wattage if this Bit is "ON"*)
	MinSP : INT;			(* Define Min SetPoint Input, if SP set below this value, the PV will become "0"*)
	MaxSP : INT;			(* Define Max SetPoint Input, if SP set Greater than value, the PV will become "0"*)
	MaxWatt : INT;		(* Defined Max Watt of Generator, Usually is 700W*)


END_VAR

VAR_OUTPUT

	iAI1raw : INT;			(*1st Raw Data to feed to Analog Output Card for Ultrasonic Generator Power Control*)
	iAI2raw : INT;			(*2nd Raw Data to feed to Analog Output Card for Ultrasonic Generator Power Control*)
	iAI3raw : INT;			(*3rd Raw Data to feed to Analog Output Card for Ultrasonic Generator Power Control*)
	iAI4raw : INT;			(*4th Raw Data to feed to Analog Output Card for Ultrasonic Generator Power Control*)
	iAI5raw : INT;			(*5th Raw Data to feed to Analog Output Card for Ultrasonic Generator Power Control*)
	iAI6raw : INT;			(*6th Raw Data to feed to Analog Output Card for Ultrasonic Generator Power Control*)

END_VAR
VAR
	iAI1f: LREAL;
	iAI2f: LREAL;
	iAI3f: LREAL;
	iAI4f: LREAL;
	iAI5f: LREAL;
	iAI6f: LREAL;

	iAI1_Wf: LREAL;
	iAI2_Wf: LREAL;
	iAI3_Wf: LREAL;
	iAI4_Wf: LREAL;
	iAI5_Wf: LREAL;
	iAI6_Wf: LREAL;

	n : INT;
	WRatio: INT;
END_VAR

(*Set Min and Max Limit for Watt input*)
(*Convert INT to LREAL for Calculation*)

IF iAI1SP>=MinSP AND iAI1SP<=MaxSP THEN
iAI1_Wf := INT_TO_LREAL (iAI1SP);
ELSE iAI1_Wf := 0;
END_IF

IF iAI2SP>=MinSP AND iAI2SP<=MaxSP THEN
iAI2_Wf := INT_TO_LREAL (iAI2SP);
ELSE iAI2_Wf := 0;
END_IF

IF iAI3SP>=MinSP AND iAI3SP<=MaxSP THEN
iAI3_Wf := INT_TO_LREAL (iAI3SP);
ELSE iAI3_Wf := 0;
END_IF

IF iAI4SP>=MinSP AND iAI4SP<=MaxSP THEN
iAI4_Wf := INT_TO_LREAL (iAI4SP);
ELSE iAI4_Wf := 0;
END_IF

IF iAI5SP>=MinSP AND iAI5SP<=MaxSP THEN
iAI5_Wf := INT_TO_LREAL (iAI5SP);
ELSE iAI5_Wf := 0;
END_IF

IF iAI6SP>=MinSP AND iAI6SP<=MaxSP THEN
iAI6_Wf := INT_TO_LREAL (iAI6SP);
ELSE iAI6_Wf := 0;
END_IF

(*Program to select Watt Base or Percent Base*)

IF PercentBase AND NOT WattBase THEN
n := 11;
END_IF

IF WattBase AND NOT PercentBase THEN
n := 10;
END_IF

IF NOT PercentBase AND NOT WattBase THEN
n := 0;
END_IF

IF PercentBase AND WattBase THEN
n:= 0;
END_IF



CASE n OF

0:;	(*No Calculation Apply*)

10:	(*Watt Base Calculation*)

WRatio := MaxWatt/100;


	iAI1f	:= iAI1_Wf/WRatio*327.67;
	iAI2f	:= iAI2_Wf/WRatio*327.67;
	iAI3f	:= iAI3_Wf/WRatio*327.67;
	iAI4f	:= iAI4_Wf/WRatio*327.67;
	iAI5f	:= iAI5_Wf/WRatio*327.67;
	iAI6f	:= iAI6_Wf/WRatio*327.67;


(*	iAI1f	:= (SQRT(iAI1_Wf/20))*3276.7;
	iAI2f	:= (SQRT(iAI2_Wf/20))*3276.7;
	iAI3f	:= (SQRT(iAI3_Wf/20))*3276.7;
	iAI4f	:= (SQRT(iAI4_Wf/20))*3276.7;
	iAI5f	:= (SQRT(iAI5_Wf/20))*3276.7;
	iAI6f	:= (SQRT(iAI6_Wf/20))*3276.7;
*)

11: 	(*% Base Calculation*)

	iAI1f	:= iAI1_Wf*327.67;
	iAI2f	:= iAI2_Wf*327.67;
	iAI3f	:= iAI3_Wf*327.67;
	iAI4f	:= iAI4_Wf*327.67;
	iAI5f	:= iAI5_Wf*327.67;
	iAI6f	:= iAI6_Wf*327.67;

END_CASE

iAI1raw := LREAL_TO_INT (iAI1f);
iAI2raw := LREAL_TO_INT (iAI2f);
iAI3raw := LREAL_TO_INT (iAI3f);
iAI4raw := LREAL_TO_INT (iAI4f);
iAI5raw := LREAL_TO_INT (iAI5f);
iAI6raw := LREAL_TO_INT (iAI6f);

END_FUNCTION_BLOCK

